BEGIN
	(*
	----------------------------------------------------------------------------------------
	|                                                                                      |
	|  Copyright  2023             FORTNA Europe BV                                        |
	|  All Rights Reserved         Netherlands                                             |
	|                                                                                      |
	----------------------------------------------------------------------------------------

	Version history:
	Date        | Version   | Author          | Remark
	----------------------------------------------------------------------------------------
	22/3/2022   | 0.1       | R. Golonka      | Unloader Alarm | DHL Munich 2023
	13/3/2024   | 0.2       | S.Nieswiec      | Alligned for new baseline
	*)

	REGION 1 - Jam
	    //  Program Alarm jam
	    #Jam(SIG := #iq_UDT_UnloaderStatus.Specific.PEC_EoS.Jam,
	         TIMESTAMP := #Time,
	         SD_1 := #is_ID);
	END_REGION

	REGION 2 - Disabled
	    //  Program Alarm disabled
	    #Disabled(SIG := #iq_UDT_UnloaderStatus.Specific.Disabled,
	              TIMESTAMP := #Time,
	              SD_1 := #is_ID);
	END_REGION

	REGION 3 - Too Long Parcel
	    //  Program Alarm too long parcel
	    #TooLongParcel(SIG := #iq_UDT_UnloaderStatus.Specific.TooLongParcel,
	                   TIMESTAMP := #Time,
	                   SD_1 := #is_ID);
	END_REGION

	REGION 4 - VFD Error
	    //  Program Alarm VFD Error
	    #VFDError(SIG := #iq_UDT_UnloaderStatus.Specific.VFDError,
	              TIMESTAMP := #Time,
	              SD_1 := #is_ID);
	END_REGION

	REGION 5 - Not healthy
	    //  Program Alarm not healthy
	    #NotHealthy(SIG := #iq_UDT_UnloaderStatus.Specific.NotHealthy,
	                TIMESTAMP := #Time,
	                SD_1 := #is_ID);
	END_REGION

END_FUNCTION_BLOCK

FUNCTION_BLOCK "FB_TP_ALARM_RIO"
{ S7_Optimized_Access := 'TRUE' }
VERSION : 0.1
// ATTRIBUTES
// AUTO_NUMBER = True
// BLOCK_NUMBER = 191
// END_ATTRIBUTES
   VAR_INPUT
      "Time" {InstructionName := 'DTL'; LibVersion := '1.0'; ExternalAccessible := 'False'; ExternalVisible := 'False'; ExternalWritable := 'False'} : DTL;   // Actual Time
      is_ID { ExternalAccessible := 'False'; ExternalVisible := 'False'; ExternalWritable := 'False'} : String;   // ID of component
   END_VAR

   VAR_IN_OUT
      iq_UDT_RIOStatus : "UDT_RIOStatus";   // Rio Status
   END_VAR

   VAR
      PNSlaveNotOnline {InstructionName := 'Program_Alarm'; LibVersion := '1.0'; ExternalAccessible := 'False'; ExternalVisible := 'False'; ExternalWritable := 'False'; S7_SetPoint := 'False'} : Program_Alarm;   // Program alarm profinet slave not online
      PNSlaveError {InstructionName := 'Program_Alarm'; LibVersion := '1.0'; ExternalAccessible := 'False'; ExternalVisible := 'False'; ExternalWritable := 'False'; S7_SetPoint := 'False'} : Program_Alarm;   // Program alarm profinet slave error
      ET200sp_ErrorModule {InstructionName := 'Program_Alarm'; LibVersion := '1.0'; ExternalAccessible := 'False'; ExternalVisible := 'False'; ExternalWritable := 'False'; S7_SetPoint := 'False'} : Array[0..31] of Program_Alarm;   // Program alarm ET200sp module error
      PNSlaveWarning {InstructionName := 'Program_Alarm'; LibVersion := '1.0'; ExternalAccessible := 'False'; ExternalVisible := 'False'; ExternalWritable := 'False'; S7_SetPoint := 'False'} : Program_Alarm;   // Program alarm profinet slave warning
   END_VAR

   VAR_TEMP
      ti_NrOfArrayEl : Int;   // Number of array element
      ti_ArraySize : Int;   // Array size
   END_VAR


BEGIN
	(*
	----------------------------------------------------------------------------------------
	|                                                                                      |
	|  Copyright  2023             FORTNA Europe BV                                        |
	|  All Rights Reserved         Netherlands                                             |
	|                                                                                      |
	----------------------------------------------------------------------------------------

	Version history:
	Date        | Version   | Author          | Remark
	----------------------------------------------------------------------------------------
	22/03/2023  | 0.1       | R. Golonka      | RIO Alarm | DHL Munich 2023
	13/3/2024   | 0.2       | S.Nieswiec      | Alligned for new baseline
	*)
	REGION 1 - Profinet slave not online
	    // Program alarm profinet slave not online
	    #PNSlaveNotOnline(SIG := #iq_UDT_RIOStatus.Specific.PNSlaveNotOnline,
	                      TIMESTAMP := #Time,
	                      SD_1 := #is_ID);
	END_REGION

	REGION 2 - Profinet slave error
	    // Program alarm profinet slave error
	    #PNSlaveError(SIG := #iq_UDT_RIOStatus.Specific.PNSlaveError,
	                  TIMESTAMP := #Time,
	                  SD_1 := #is_ID);
	END_REGION

	REGION 3 - Profinet slave warning
	    // Program alarm profinet slave warning
	    #PNSlaveWarning(SIG := #iq_UDT_RIOStatus.Specific.PNSlaveWarning,
	                    TIMESTAMP := #Time,
	                    SD_1 := #is_ID);
	END_REGION

	REGION 4 - ET200SP module error
	    // Array size
	    #ti_ArraySize := "FC_GetNrOfArrayEl"(#iq_UDT_RIOStatus.Specific.ET200sp_ErrorModule);

	    // Program alarm ET200SP module error
	    FOR #ti_NrOfArrayEl := 0 TO (#ti_ArraySize - 1) DO
	        #ET200sp_ErrorModule[#ti_NrOfArrayEl](SIG := #iq_UDT_RIOStatus.Specific.ET200sp_ErrorModule[#ti_NrOfArrayEl],
	                                              TIMESTAMP := #Time,
	                                              SD_1 := #is_ID);
	    END_FOR;
	END_REGION
END_FUNCTION_BLOCK

FUNCTION_BLOCK "FB_TP_ALARM_RetractableRoller"
{ S7_Optimized_Access := 'TRUE' }
VERSION : 0.1
// ATTRIBUTES
// AUTO_NUMBER = True
// BLOCK_NUMBER = 190
// END_ATTRIBUTES
   VAR_INPUT
      "Time" { ExternalAccessible := 'False'; ExternalVisible := 'False'; ExternalWritable := 'False'} : LDT;   // Actual Time
      is_ID { ExternalAccessible := 'False'; ExternalVisible := 'False'; ExternalWritable := 'False'} : String;   // ID of component
   END_VAR

   VAR_IN_OUT
      iq_UDT_RetractableRollerStatus : "UDT_RetractrableRoller_Status";
   END_VAR

   VAR
      NoHomePosition {InstructionName := 'Program_Alarm'; LibVersion := '1.0'; ExternalAccessible := 'False'; ExternalVisible := 'False'; ExternalWritable := 'False'; S7_SetPoint := 'False'} : Program_Alarm;
      RollerError {InstructionName := 'Program_Alarm'; LibVersion := '1.0'; ExternalAccessible := 'False'; ExternalVisible := 'False'; ExternalWritable := 'False'; S7_SetPoint := 'False'} : Program_Alarm;
   END_VAR


BEGIN
	(*
	----------------------------------------------------------------------------------------
	|                                                                                      |
	|  Copyright  2023             FORTNA Europe BV                                        |
	|  All Rights Reserved         Netherlands                                             |
	|                                                                                      |
	----------------------------------------------------------------------------------------

	Version history:
	Date        | Version   | Author          | Remark
	----------------------------------------------------------------------------------------
	09/05/2023   | 0.1       | M. Diebel       | ABSwitch Alarm | DHL Munich 2023
	13/3/2024    | 0.2       | S.Nieswiec      | Alligned for new baseline
	*)

	REGION 1 - NoHomePosition
	    //Program Alarm NoHomePosition
	    #NoHomePosition(SIG := #iq_UDT_RetractableRollerStatus.Specific.NoHomePosition,
	                    TIMESTAMP := #Time,
	                    SD_1 := #is_ID);
	END_REGION

	REGION 2 - RollerError
	    //Program Alarm RollerError
	    #RollerError(SIG := #iq_UDT_RetractableRollerStatus.Specific.RollerError,
	                 TIMESTAMP := #Time,
	                 SD_1 := #is_ID);
	END_REGION
END_FUNCTION_BLOCK

FUNCTION_BLOCK "FB_TP_ALARM_Rapiscan"
{ S7_Optimized_Access := 'TRUE' }
VERSION : 0.1
// ATTRIBUTES
// AUTO_NUMBER = True
// BLOCK_NUMBER = 189
// END_ATTRIBUTES
   VAR_INPUT
      "Time" { ExternalAccessible := 'False'; ExternalVisible := 'False'; ExternalWritable := 'False'} : LDT;   // Actual Time
      is_ID { ExternalAccessible := 'False'; ExternalVisible := 'False'; ExternalWritable := 'False'} : String;   // ID of component
   END_VAR

   VAR_IN_OUT
      iq_UDT_RapiscanStatus : "UDT_RapiscanStatus";   // Rapiscan Status
   END_VAR

   VAR
      XrayEnergised {InstructionName := 'Program_Alarm'; LibVersion := '1.0'; ExternalAccessible := 'False'; ExternalVisible := 'False'; ExternalWritable := 'False'; S7_SetPoint := 'False'} : Program_Alarm;   // Program Alarm Xray energised error
      XrayFault {InstructionName := 'Program_Alarm'; LibVersion := '1.0'; ExternalAccessible := 'False'; ExternalVisible := 'False'; ExternalWritable := 'False'; S7_SetPoint := 'False'} : Program_Alarm;   // Program Alarm Xray foult error
      XrayRdyRCV {InstructionName := 'Program_Alarm'; LibVersion := '1.0'; ExternalAccessible := 'False'; ExternalVisible := 'False'; ExternalWritable := 'False'; S7_SetPoint := 'False'} : Program_Alarm;   // Program Alarm Xray ready recieve info
      XrayRdySend {InstructionName := 'Program_Alarm'; LibVersion := '1.0'; ExternalAccessible := 'False'; ExternalVisible := 'False'; ExternalWritable := 'False'; S7_SetPoint := 'False'} : Program_Alarm;   // Program Alarm Xray ready send info
      BagScanning {InstructionName := 'Program_Alarm'; LibVersion := '1.0'; ExternalAccessible := 'False'; ExternalVisible := 'False'; ExternalWritable := 'False'; S7_SetPoint := 'False'} : Program_Alarm;   // Program Alarm bag scanming info
      TransportMode {InstructionName := 'Program_Alarm'; LibVersion := '1.0'; ExternalAccessible := 'False'; ExternalVisible := 'False'; ExternalWritable := 'False'; S7_SetPoint := 'False'} : Program_Alarm;   // Program Alarm transport mode info
      BackBelt {InstructionName := 'Program_Alarm'; LibVersion := '1.0'; ExternalAccessible := 'False'; ExternalVisible := 'False'; ExternalWritable := 'False'; S7_SetPoint := 'False'} : Program_Alarm;   // Program Alarm backbelt info
   END_VAR


BEGIN
	(*
	----------------------------------------------------------------------------------------
	|                                                                                      |
	|  Copyright  2023             FORTNA Europe BV                                        |
	|  All Rights Reserved         Netherlands                                             |
	|                                                                                      |
	----------------------------------------------------------------------------------------

	Version history:
	Date        | Version   | Author          | Remark
	----------------------------------------------------------------------------------------
	25/4/2022   | 1.0       | M. Diebel       | Rapiscan Alarm | DHL Munich 2023
	13/3/2024   | 1.1       | S.Nieswiec      | Alligned for new baseline
	*)

	REGION 1 - XrayEnergised
	    //Program Alarm Xray energised error
	    #XrayEnergised(SIG := #iq_UDT_RapiscanStatus.XraySpecific.XrayEnergised,
	                   TIMESTAMP := #Time,
	                   SD_1 := #is_ID);
	END_REGION

	REGION 2 - XrayFault
	    //Program Alarm Xray foult error
	    #XrayFault(SIG := #iq_UDT_RapiscanStatus.XraySpecific.XrayFault,
	               TIMESTAMP := #Time,
	               SD_1 := #is_ID);
	END_REGION

	REGION 3 - XrayRdyRCV
	    //Program Alarm Xray ready recieve info
	    #XrayRdyRCV(SIG := #iq_UDT_RapiscanStatus.XraySpecific.XrayRdyRCV,
	                TIMESTAMP := #Time,
	                SD_1 := #is_ID);
	END_REGION

	REGION 4 - XrayRdySend
	    //Program Alarm Xray ready send info
	    #XrayRdySend(SIG := #iq_UDT_RapiscanStatus.XraySpecific.XrayRdySend,
	                 TIMESTAMP := #Time,
	                 SD_1 := #is_ID);
	END_REGION

	REGION 5 - BagScanning
	    //Program Alarm bag scanming info
	    #BagScanning(SIG := #iq_UDT_RapiscanStatus.XraySpecific.BagScanning,
	                 TIMESTAMP := #Time,
	                 SD_1 := #is_ID);
	END_REGION

	REGION 6 - TransportMode
	    //Program Alarm transport mode info
	    #TransportMode(SIG := #iq_UDT_RapiscanStatus.XraySpecific.TransportMode,
	                   TIMESTAMP := #Time,
	                   SD_1 := #is_ID);
	END_REGION

	REGION 7 - BackBelt
	    //Program Alarm backbelt info
	    #BackBelt(SIG := #iq_UDT_RapiscanStatus.XraySpecific.BackBelt,
	              TIMESTAMP := #Time,
	              SD_1 := #is_ID);
	END_REGION



END_FUNCTION_BLOCK

FUNCTION_BLOCK "FB_TP_ALARM_PNNode"
{ S7_Optimized_Access := 'TRUE' }
VERSION : 0.1
// ATTRIBUTES
// AUTO_NUMBER = True
// BLOCK_NUMBER = 188
// END_ATTRIBUTES
   VAR_INPUT
      "Time" {InstructionName := 'DTL'; LibVersion := '1.0'; ExternalAccessible := 'False'; ExternalVisible := 'False'; ExternalWritable := 'False'} : DTL;   // Actual Time
      is_ID { ExternalAccessible := 'False'; ExternalVisible := 'False'; ExternalWritable := 'False'} : String;   // ID of component
   END_VAR

   VAR_IN_OUT
      iq_UDT_PNNode_Status : "UDT_PNNodeStatus";   // PNNode Status
   END_VAR

   VAR
      PNSlaveNotOnline {InstructionName := 'Program_Alarm'; LibVersion := '1.0'; ExternalAccessible := 'False'; ExternalVisible := 'False'; ExternalWritable := 'False'; S7_SetPoint := 'False'} : Program_Alarm;   // Program alarm profinet slave net online
      PNSlaveError {InstructionName := 'Program_Alarm'; LibVersion := '1.0'; ExternalAccessible := 'False'; ExternalVisible := 'False'; ExternalWritable := 'False'; S7_SetPoint := 'False'} : Program_Alarm;   // Program alarm profinet slave error
      PNSlaveWarning {InstructionName := 'Program_Alarm'; LibVersion := '1.0'; ExternalAccessible := 'False'; ExternalVisible := 'False'; ExternalWritable := 'False'; S7_SetPoint := 'False'} : Program_Alarm;   // Program alarm profinet slave warning
   END_VAR


BEGIN
	(*
	----------------------------------------------------------------------------------------
	|                                                                                      |
	|  Copyright  2023             FORTNA Europe BV                                        |
	|  All Rights Reserved         Netherlands                                             |
	|                                                                                      |
	----------------------------------------------------------------------------------------

	Version history:
	Date        | Version   | Author          | Remark
	----------------------------------------------------------------------------------------
	22/03/2023  | 0.1       | R. Golonka      | PN Node Alarm | DHL Munich 2023
	13/3/2024   | 0.2       | S.Nieswiec      | Alligned for new baseline
	*)

	REGION 1 - Profinet slave not online
	    // Program Alarm profinet slave not online
	    #PNSlaveNotOnline(SIG := #iq_UDT_PNNode_Status.Specific.PNSlaveNotOnline,
	                      TIMESTAMP := #Time,
	                      SD_1 := #is_ID);
	END_REGION

	REGION 2 - Profinet slave error
	    // Program Alarm profinet slave error
	    #PNSlaveError(SIG := #iq_UDT_PNNode_Status.Specific.PNSlaveError,
	                  TIMESTAMP := #Time,
	                  SD_1 := #is_ID);
	END_REGION

	REGION 3 - Profinet slave warning
	    // Program Alarm profinet slave warning
	    #PNSlaveWarning(SIG := #iq_UDT_PNNode_Status.Specific.PNSlaveWarning,
	                    TIMESTAMP := #Time,
	                    SD_1 := #is_ID);
	END_REGION
END_FUNCTION_BLOCK

FUNCTION_BLOCK "FB_TP_ALARM_PECUpdate"
{ S7_Optimized_Access := 'TRUE' }
VERSION : 0.1
// ATTRIBUTES
// AUTO_NUMBER = True
// BLOCK_NUMBER = 187
// END_ATTRIBUTES
   VAR_INPUT
      "Time" {InstructionName := 'DTL'; LibVersion := '1.0'; ExternalAccessible := 'False'; ExternalVisible := 'False'; ExternalWritable := 'False'} : DTL;   // Actual Time
      is_ID { ExternalAccessible := 'False'; ExternalVisible := 'False'; ExternalWritable := 'False'} : String;   // ID of component
   END_VAR

   VAR_IN_OUT
      iq_UDT_PECUpdate_Status : "UDT_PECUpdateStatus";   // PEC Update Status
   END_VAR

   VAR
      Jam {InstructionName := 'Program_Alarm'; LibVersion := '1.0'; ExternalAccessible := 'False'; ExternalVisible := 'False'; ExternalWritable := 'False'; S7_SetPoint := 'False'} : Program_Alarm;   // Program Alarm Jam
      TooManyLost {InstructionName := 'Program_Alarm'; LibVersion := '1.0'; ExternalAccessible := 'False'; ExternalVisible := 'False'; ExternalWritable := 'False'; S7_SetPoint := 'False'} : Program_Alarm;   // Program Alarm Too many losy
      LowPerformance {InstructionName := 'Program_Alarm'; LibVersion := '1.0'; ExternalAccessible := 'False'; ExternalVisible := 'False'; ExternalWritable := 'False'; S7_SetPoint := 'False'} : Program_Alarm;   // Program Alarm Low performance
   END_VAR


BEGIN
	(*
	----------------------------------------------------------------------------------------
	|                                                                                      |
	|  Copyright  2023             FORTNA Europe BV                                        |
	|  All Rights Reserved         Netherlands                                             |
	|                                                                                      |
	----------------------------------------------------------------------------------------

	Version history:
	Date        | Version   | Author          | Remark
	----------------------------------------------------------------------------------------
	22/3/2022   | 0.1       | R. Golonka      | PEC Update Alarm | DHL Munich 2023
	13/3/2024   | 0.2       | S.Nieswiec      | Alligned for new baseline
	*)

	REGION 1- Jam
	    // Program Alarm Jam
	    #Jam(SIG := #iq_UDT_PECUpdate_Status.Jam,
	         TIMESTAMP := #Time,
	         SD_1 := #is_ID);
	END_REGION

	REGION 2 - Too many lost
	    // Program Alarm Too many losy
	    #TooManyLost(SIG := #iq_UDT_PECUpdate_Status.TooManyLost,
	                 TIMESTAMP := #Time,
	                 SD_1 := #is_ID);
	END_REGION

	REGION 3 - Low Performance
	    // Program Alarm Low performance
	    #LowPerformance(SIG := #iq_UDT_PECUpdate_Status.LowPerformance,
	                    TIMESTAMP := #Time,
	                    SD_1 := #is_ID);
	END_REGION

END_FUNCTION_BLOCK

FUNCTION_BLOCK "FB_TP_ALARM_PEC"
{ S7_Optimized_Access := 'TRUE' }
VERSION : 0.1
// ATTRIBUTES
// AUTO_NUMBER = True
// BLOCK_NUMBER = 186
// END_ATTRIBUTES
   VAR_INPUT
      "Time" {InstructionName := 'DTL'; LibVersion := '1.0'; ExternalAccessible := 'False'; ExternalVisible := 'False'; ExternalWritable := 'False'} : DTL;   // Actual Time
      is_ID { ExternalAccessible := 'False'; ExternalVisible := 'False'; ExternalWritable := 'False'} : String;   // ID of component
   END_VAR

   VAR_IN_OUT
      iq_UDT_PEC_Status : "UDT_PECStatus";   // PEC Status
   END_VAR

   VAR
      Jam {InstructionName := 'Program_Alarm'; LibVersion := '1.0'; ExternalAccessible := 'False'; ExternalVisible := 'False'; ExternalWritable := 'False'; S7_SetPoint := 'False'} : Program_Alarm;   // Program Alarm Jam
   END_VAR


BEGIN
	(*
	----------------------------------------------------------------------------------------
	|                                                                                      |
	|  Copyright  2023             FORTNA Europe BV                                        |
	|  All Rights Reserved         Netherlands                                             |
	|                                                                                      |
	----------------------------------------------------------------------------------------

	Version history:
	Date        | Version   | Author          | Remark
	----------------------------------------------------------------------------------------
	22/3/2022   | 0.1       | R. Golonka      | PEC Alarm | DHL Munich 2023
	13/3/2024   | 0.2       | S.Nieswiec      | Alligned for new baseline
	*)

	REGION 1- Jam
	    // Program Alarm Jam
	    #Jam(SIG := #iq_UDT_PEC_Status.Jam,
	         TIMESTAMP := #Time,
	         SD_1 := #is_ID);
	END_REGION


END_FUNCTION_BLOCK

FUNCTION_BLOCK "FB_TP_ALARM_PDP"
{ S7_Optimized_Access := 'TRUE' }
VERSION : 0.1
// ATTRIBUTES
// AUTO_NUMBER = True
// BLOCK_NUMBER = 185
// END_ATTRIBUTES
   VAR_INPUT
      "Time" { ExternalAccessible := 'False'; ExternalVisible := 'False'; ExternalWritable := 'False'} : LDT;   // Actual Time
      is_ID { ExternalAccessible := 'False'; ExternalVisible := 'False'; ExternalWritable := 'False'} : String;   // ID of component
   END_VAR

   VAR_IN_OUT
      iq_UDT_PDPStatus : "UDT_PDPStatus";   // PDP Status
   END_VAR

   VAR
      CircuitBreakersTripped {InstructionName := 'Program_Alarm'; LibVersion := '1.0'; ExternalAccessible := 'False'; ExternalVisible := 'False'; ExternalWritable := 'False'; S7_SetPoint := 'False'} : Program_Alarm;   // Program Alarm circuit breakers tripped
      CircuitBreakerStateF100_F200_F300 {InstructionName := 'Program_Alarm'; LibVersion := '1.0'; ExternalAccessible := 'False'; ExternalVisible := 'False'; ExternalWritable := 'False'; S7_SetPoint := 'False'} : Program_Alarm;   // Program Alarm circuit breakers state
      CircuitBreakerStatePM {InstructionName := 'Program_Alarm'; LibVersion := '1.0'; ExternalAccessible := 'False'; ExternalVisible := 'False'; ExternalWritable := 'False'; S7_SetPoint := 'False'} : Program_Alarm;   // Program Alarm circuit breakers state PM
      CircuitBreakerTrippedF101 {InstructionName := 'Program_Alarm'; LibVersion := '1.0'; ExternalAccessible := 'False'; ExternalVisible := 'False'; ExternalWritable := 'False'; S7_SetPoint := 'False'} : Program_Alarm;   // Program Alarm circuit breakers tripped
      CircuitBreakerTrippedF102 {InstructionName := 'Program_Alarm'; LibVersion := '1.0'; ExternalAccessible := 'False'; ExternalVisible := 'False'; ExternalWritable := 'False'; S7_SetPoint := 'False'} : Program_Alarm;   // Program Alarm circuit breakers tripped
      CircuitBreakerTrippedF103 {InstructionName := 'Program_Alarm'; LibVersion := '1.0'; ExternalAccessible := 'False'; ExternalVisible := 'False'; ExternalWritable := 'False'; S7_SetPoint := 'False'} : Program_Alarm;   // Program Alarm circuit breakers tripped
      CircuitBreakerTrippedF104 {InstructionName := 'Program_Alarm'; LibVersion := '1.0'; ExternalAccessible := 'False'; ExternalVisible := 'False'; ExternalWritable := 'False'; S7_SetPoint := 'False'} : Program_Alarm;   // Program Alarm circuit breakers tripped
      CircuitBreakerTrippedF105 {InstructionName := 'Program_Alarm'; LibVersion := '1.0'; ExternalAccessible := 'False'; ExternalVisible := 'False'; ExternalWritable := 'False'; S7_SetPoint := 'False'} : Program_Alarm;   // Program Alarm circuit breakers tripped
      CircuitBreakerTrippedF106 {InstructionName := 'Program_Alarm'; LibVersion := '1.0'; ExternalAccessible := 'False'; ExternalVisible := 'False'; ExternalWritable := 'False'; S7_SetPoint := 'False'} : Program_Alarm;   // Program Alarm circuit breakers tripped
      CircuitBreakerTrippedF107 {InstructionName := 'Program_Alarm'; LibVersion := '1.0'; ExternalAccessible := 'False'; ExternalVisible := 'False'; ExternalWritable := 'False'; S7_SetPoint := 'False'} : Program_Alarm;   // Program Alarm circuit breakers tripped
      CircuitBreakerTrippedF108 {InstructionName := 'Program_Alarm'; LibVersion := '1.0'; ExternalAccessible := 'False'; ExternalVisible := 'False'; ExternalWritable := 'False'; S7_SetPoint := 'False'} : Program_Alarm;   // Program Alarm circuit breakers tripped
      CircuitBreakerTrippedF109 {InstructionName := 'Program_Alarm'; LibVersion := '1.0'; ExternalAccessible := 'False'; ExternalVisible := 'False'; ExternalWritable := 'False'; S7_SetPoint := 'False'} : Program_Alarm;   // Program Alarm circuit breakers tripped
      CircuitBreakerTrippedF110 {InstructionName := 'Program_Alarm'; LibVersion := '1.0'; ExternalAccessible := 'False'; ExternalVisible := 'False'; ExternalWritable := 'False'; S7_SetPoint := 'False'} : Program_Alarm;   // Program Alarm circuit breakers tripped
      CircuitBreakerTrippedF111 {InstructionName := 'Program_Alarm'; LibVersion := '1.0'; ExternalAccessible := 'False'; ExternalVisible := 'False'; ExternalWritable := 'False'; S7_SetPoint := 'False'} : Program_Alarm;   // Program Alarm circuit breakers tripped
      CircuitBreakerTrippedF112 {InstructionName := 'Program_Alarm'; LibVersion := '1.0'; ExternalAccessible := 'False'; ExternalVisible := 'False'; ExternalWritable := 'False'; S7_SetPoint := 'False'} : Program_Alarm;   // Program Alarm circuit breakers tripped
      CircuitBreakerTrippedF113 {InstructionName := 'Program_Alarm'; LibVersion := '1.0'; ExternalAccessible := 'False'; ExternalVisible := 'False'; ExternalWritable := 'False'; S7_SetPoint := 'False'} : Program_Alarm;   // Program Alarm circuit breakers tripped
      CircuitBreakerTrippedF114 {InstructionName := 'Program_Alarm'; LibVersion := '1.0'; ExternalAccessible := 'False'; ExternalVisible := 'False'; ExternalWritable := 'False'; S7_SetPoint := 'False'} : Program_Alarm;   // Program Alarm circuit breakers tripped
      CircuitBreakerTrippedF115 {InstructionName := 'Program_Alarm'; LibVersion := '1.0'; ExternalAccessible := 'False'; ExternalVisible := 'False'; ExternalWritable := 'False'; S7_SetPoint := 'False'} : Program_Alarm;   // Program Alarm circuit breakers tripped
      CircuitBreakerTrippedF116 {InstructionName := 'Program_Alarm'; LibVersion := '1.0'; ExternalAccessible := 'False'; ExternalVisible := 'False'; ExternalWritable := 'False'; S7_SetPoint := 'False'} : Program_Alarm;   // Program Alarm circuit breakers tripped
      CircuitBreakerTrippedF117 {InstructionName := 'Program_Alarm'; LibVersion := '1.0'; ExternalAccessible := 'False'; ExternalVisible := 'False'; ExternalWritable := 'False'; S7_SetPoint := 'False'} : Program_Alarm;   // Program Alarm circuit breakers tripped
      CircuitBreakerTrippedF118 {InstructionName := 'Program_Alarm'; LibVersion := '1.0'; ExternalAccessible := 'False'; ExternalVisible := 'False'; ExternalWritable := 'False'; S7_SetPoint := 'False'} : Program_Alarm;   // Program Alarm circuit breakers tripped
      CircuitBreakerTrippedF119 {InstructionName := 'Program_Alarm'; LibVersion := '1.0'; ExternalAccessible := 'False'; ExternalVisible := 'False'; ExternalWritable := 'False'; S7_SetPoint := 'False'} : Program_Alarm;   // Program Alarm circuit breakers tripped
      CircuitBreakerTrippedF120 {InstructionName := 'Program_Alarm'; LibVersion := '1.0'; ExternalAccessible := 'False'; ExternalVisible := 'False'; ExternalWritable := 'False'; S7_SetPoint := 'False'} : Program_Alarm;   // Program Alarm circuit breakers tripped
      CircuitBreakerTrippedF121 {InstructionName := 'Program_Alarm'; LibVersion := '1.0'; ExternalAccessible := 'False'; ExternalVisible := 'False'; ExternalWritable := 'False'; S7_SetPoint := 'False'} : Program_Alarm;   // Program Alarm circuit breakers tripped
      CircuitBreakerTrippedF122 {InstructionName := 'Program_Alarm'; LibVersion := '1.0'; ExternalAccessible := 'False'; ExternalVisible := 'False'; ExternalWritable := 'False'; S7_SetPoint := 'False'} : Program_Alarm;   // Program Alarm circuit breakers tripped
      CircuitBreakerTrippedF123 {InstructionName := 'Program_Alarm'; LibVersion := '1.0'; ExternalAccessible := 'False'; ExternalVisible := 'False'; ExternalWritable := 'False'; S7_SetPoint := 'False'} : Program_Alarm;   // Program Alarm circuit breakers tripped
      CircuitBreakerTrippedF124 {InstructionName := 'Program_Alarm'; LibVersion := '1.0'; ExternalAccessible := 'False'; ExternalVisible := 'False'; ExternalWritable := 'False'; S7_SetPoint := 'False'} : Program_Alarm;   // Program Alarm circuit breakers tripped
      CircuitBreakerTrippedF125 {InstructionName := 'Program_Alarm'; LibVersion := '1.0'; ExternalAccessible := 'False'; ExternalVisible := 'False'; ExternalWritable := 'False'; S7_SetPoint := 'False'} : Program_Alarm;   // Program Alarm circuit breakers tripped
      CircuitBreakerTrippedF126 {InstructionName := 'Program_Alarm'; LibVersion := '1.0'; ExternalAccessible := 'False'; ExternalVisible := 'False'; ExternalWritable := 'False'; S7_SetPoint := 'False'} : Program_Alarm;   // Program Alarm circuit breakers tripped
      CircuitBreakerTrippedF127 {InstructionName := 'Program_Alarm'; LibVersion := '1.0'; ExternalAccessible := 'False'; ExternalVisible := 'False'; ExternalWritable := 'False'; S7_SetPoint := 'False'} : Program_Alarm;   // Program Alarm circuit breakers tripped
      CircuitBreakerTrippedF128 {InstructionName := 'Program_Alarm'; LibVersion := '1.0'; ExternalAccessible := 'False'; ExternalVisible := 'False'; ExternalWritable := 'False'; S7_SetPoint := 'False'} : Program_Alarm;   // Program Alarm circuit breakers tripped
      CircuitBreakerTrippedF129 {InstructionName := 'Program_Alarm'; LibVersion := '1.0'; ExternalAccessible := 'False'; ExternalVisible := 'False'; ExternalWritable := 'False'; S7_SetPoint := 'False'} : Program_Alarm;   // Program Alarm circuit breakers tripped
      CircuitBreakerTrippedF130 {InstructionName := 'Program_Alarm'; LibVersion := '1.0'; ExternalAccessible := 'False'; ExternalVisible := 'False'; ExternalWritable := 'False'; S7_SetPoint := 'False'} : Program_Alarm;   // Program Alarm circuit breakers tripped
      CircuitBreakerTrippedF131 {InstructionName := 'Program_Alarm'; LibVersion := '1.0'; ExternalAccessible := 'False'; ExternalVisible := 'False'; ExternalWritable := 'False'; S7_SetPoint := 'False'} : Program_Alarm;   // Program Alarm circuit breakers tripped
      CircuitBreakerTrippedF132 {InstructionName := 'Program_Alarm'; LibVersion := '1.0'; ExternalAccessible := 'False'; ExternalVisible := 'False'; ExternalWritable := 'False'; S7_SetPoint := 'False'} : Program_Alarm;   // Program Alarm circuit breakers tripped
      CircuitBreakerTrippedF133 {InstructionName := 'Program_Alarm'; LibVersion := '1.0'; ExternalAccessible := 'False'; ExternalVisible := 'False'; ExternalWritable := 'False'; S7_SetPoint := 'False'} : Program_Alarm;   // Program Alarm circuit breakers tripped
      CircuitBreakerTrippedF134 {InstructionName := 'Program_Alarm'; LibVersion := '1.0'; ExternalAccessible := 'False'; ExternalVisible := 'False'; ExternalWritable := 'False'; S7_SetPoint := 'False'} : Program_Alarm;   // Program Alarm circuit breakers tripped
      CircuitBreakerTrippedF135 {InstructionName := 'Program_Alarm'; LibVersion := '1.0'; ExternalAccessible := 'False'; ExternalVisible := 'False'; ExternalWritable := 'False'; S7_SetPoint := 'False'} : Program_Alarm;   // Program Alarm circuit breakers tripped
      CircuitBreakerTrippedF201 {InstructionName := 'Program_Alarm'; LibVersion := '1.0'; ExternalAccessible := 'False'; ExternalVisible := 'False'; ExternalWritable := 'False'; S7_SetPoint := 'False'} : Program_Alarm;   // Program Alarm circuit breakers tripped
      CircuitBreakerTrippedF202 {InstructionName := 'Program_Alarm'; LibVersion := '1.0'; ExternalAccessible := 'False'; ExternalVisible := 'False'; ExternalWritable := 'False'; S7_SetPoint := 'False'} : Program_Alarm;   // Program Alarm circuit breakers tripped
      CircuitBreakerTrippedF203 {InstructionName := 'Program_Alarm'; LibVersion := '1.0'; ExternalAccessible := 'False'; ExternalVisible := 'False'; ExternalWritable := 'False'; S7_SetPoint := 'False'} : Program_Alarm;   // Program Alarm circuit breakers tripped
      CircuitBreakerTrippedF204 {InstructionName := 'Program_Alarm'; LibVersion := '1.0'; ExternalAccessible := 'False'; ExternalVisible := 'False'; ExternalWritable := 'False'; S7_SetPoint := 'False'} : Program_Alarm;   // Program Alarm circuit breakers tripped
      CircuitBreakerTrippedF205 {InstructionName := 'Program_Alarm'; LibVersion := '1.0'; ExternalAccessible := 'False'; ExternalVisible := 'False'; ExternalWritable := 'False'; S7_SetPoint := 'False'} : Program_Alarm;   // Program Alarm circuit breakers tripped
      CircuitBreakerTrippedF206 {InstructionName := 'Program_Alarm'; LibVersion := '1.0'; ExternalAccessible := 'False'; ExternalVisible := 'False'; ExternalWritable := 'False'; S7_SetPoint := 'False'} : Program_Alarm;   // Program Alarm circuit breakers tripped
      CircuitBreakerTrippedF207 {InstructionName := 'Program_Alarm'; LibVersion := '1.0'; ExternalAccessible := 'False'; ExternalVisible := 'False'; ExternalWritable := 'False'; S7_SetPoint := 'False'} : Program_Alarm;   // Program Alarm circuit breakers tripped
      CircuitBreakerTrippedF208 {InstructionName := 'Program_Alarm'; LibVersion := '1.0'; ExternalAccessible := 'False'; ExternalVisible := 'False'; ExternalWritable := 'False'; S7_SetPoint := 'False'} : Program_Alarm;   // Program Alarm circuit breakers tripped
      CircuitBreakerTrippedF209 {InstructionName := 'Program_Alarm'; LibVersion := '1.0'; ExternalAccessible := 'False'; ExternalVisible := 'False'; ExternalWritable := 'False'; S7_SetPoint := 'False'} : Program_Alarm;   // Program Alarm circuit breakers tripped
      CircuitBreakerTrippedF210 {InstructionName := 'Program_Alarm'; LibVersion := '1.0'; ExternalAccessible := 'False'; ExternalVisible := 'False'; ExternalWritable := 'False'; S7_SetPoint := 'False'} : Program_Alarm;   // Program Alarm circuit breakers tripped
      CircuitBreakerTrippedF211 {InstructionName := 'Program_Alarm'; LibVersion := '1.0'; ExternalAccessible := 'False'; ExternalVisible := 'False'; ExternalWritable := 'False'; S7_SetPoint := 'False'} : Program_Alarm;   // Program Alarm circuit breakers tripped
      CircuitBreakerTrippedF212 {InstructionName := 'Program_Alarm'; LibVersion := '1.0'; ExternalAccessible := 'False'; ExternalVisible := 'False'; ExternalWritable := 'False'; S7_SetPoint := 'False'} : Program_Alarm;   // Program Alarm circuit breakers tripped
      CircuitBreakerTrippedF213 {InstructionName := 'Program_Alarm'; LibVersion := '1.0'; ExternalAccessible := 'False'; ExternalVisible := 'False'; ExternalWritable := 'False'; S7_SetPoint := 'False'} : Program_Alarm;   // Program Alarm circuit breakers tripped
      CircuitBreakerTrippedF214 {InstructionName := 'Program_Alarm'; LibVersion := '1.0'; ExternalAccessible := 'False'; ExternalVisible := 'False'; ExternalWritable := 'False'; S7_SetPoint := 'False'} : Program_Alarm;   // Program Alarm circuit breakers tripped
      CircuitBreakerTrippedF215 {InstructionName := 'Program_Alarm'; LibVersion := '1.0'; ExternalAccessible := 'False'; ExternalVisible := 'False'; ExternalWritable := 'False'; S7_SetPoint := 'False'} : Program_Alarm;   // Program Alarm circuit breakers tripped
      CircuitBreakerTrippedF216 {InstructionName := 'Program_Alarm'; LibVersion := '1.0'; ExternalAccessible := 'False'; ExternalVisible := 'False'; ExternalWritable := 'False'; S7_SetPoint := 'False'} : Program_Alarm;   // Program Alarm circuit breakers tripped
      CircuitBreakerTrippedF217 {InstructionName := 'Program_Alarm'; LibVersion := '1.0'; ExternalAccessible := 'False'; ExternalVisible := 'False'; ExternalWritable := 'False'; S7_SetPoint := 'False'} : Program_Alarm;   // Program Alarm circuit breakers tripped
      CircuitBreakerTrippedF218 {InstructionName := 'Program_Alarm'; LibVersion := '1.0'; ExternalAccessible := 'False'; ExternalVisible := 'False'; ExternalWritable := 'False'; S7_SetPoint := 'False'} : Program_Alarm;   // Program Alarm circuit breakers tripped
      CircuitBreakerTrippedF219 {InstructionName := 'Program_Alarm'; LibVersion := '1.0'; ExternalAccessible := 'False'; ExternalVisible := 'False'; ExternalWritable := 'False'; S7_SetPoint := 'False'} : Program_Alarm;   // Program Alarm circuit breakers tripped
      CircuitBreakerTrippedF220 {InstructionName := 'Program_Alarm'; LibVersion := '1.0'; ExternalAccessible := 'False'; ExternalVisible := 'False'; ExternalWritable := 'False'; S7_SetPoint := 'False'} : Program_Alarm;   // Program Alarm circuit breakers tripped
      CircuitBreakerTrippedF221 {InstructionName := 'Program_Alarm'; LibVersion := '1.0'; ExternalAccessible := 'False'; ExternalVisible := 'False'; ExternalWritable := 'False'; S7_SetPoint := 'False'} : Program_Alarm;   // Program Alarm circuit breakers tripped
      CircuitBreakerTrippedF222 {InstructionName := 'Program_Alarm'; LibVersion := '1.0'; ExternalAccessible := 'False'; ExternalVisible := 'False'; ExternalWritable := 'False'; S7_SetPoint := 'False'} : Program_Alarm;   // Program Alarm circuit breakers tripped
      CircuitBreakerTrippedF223 {InstructionName := 'Program_Alarm'; LibVersion := '1.0'; ExternalAccessible := 'False'; ExternalVisible := 'False'; ExternalWritable := 'False'; S7_SetPoint := 'False'} : Program_Alarm;   // Program Alarm circuit breakers tripped
      CircuitBreakerTrippedF224 {InstructionName := 'Program_Alarm'; LibVersion := '1.0'; ExternalAccessible := 'False'; ExternalVisible := 'False'; ExternalWritable := 'False'; S7_SetPoint := 'False'} : Program_Alarm;   // Program Alarm circuit breakers tripped
      CircuitBreakerTrippedF225 {InstructionName := 'Program_Alarm'; LibVersion := '1.0'; ExternalAccessible := 'False'; ExternalVisible := 'False'; ExternalWritable := 'False'; S7_SetPoint := 'False'} : Program_Alarm;   // Program Alarm circuit breakers tripped
      CircuitBreakerTrippedF226 {InstructionName := 'Program_Alarm'; LibVersion := '1.0'; ExternalAccessible := 'False'; ExternalVisible := 'False'; ExternalWritable := 'False'; S7_SetPoint := 'False'} : Program_Alarm;   // Program Alarm circuit breakers tripped
      CircuitBreakerTrippedF227 {InstructionName := 'Program_Alarm'; LibVersion := '1.0'; ExternalAccessible := 'False'; ExternalVisible := 'False'; ExternalWritable := 'False'; S7_SetPoint := 'False'} : Program_Alarm;   // Program Alarm circuit breakers tripped
      CircuitBreakerTrippedF228 {InstructionName := 'Program_Alarm'; LibVersion := '1.0'; ExternalAccessible := 'False'; ExternalVisible := 'False'; ExternalWritable := 'False'; S7_SetPoint := 'False'} : Program_Alarm;   // Program Alarm circuit breakers tripped
      CircuitBreakerTrippedF229 {InstructionName := 'Program_Alarm'; LibVersion := '1.0'; ExternalAccessible := 'False'; ExternalVisible := 'False'; ExternalWritable := 'False'; S7_SetPoint := 'False'} : Program_Alarm;   // Program Alarm circuit breakers tripped
      CircuitBreakerTrippedF501 {InstructionName := 'Program_Alarm'; LibVersion := '1.0'; ExternalAccessible := 'False'; ExternalVisible := 'False'; ExternalWritable := 'False'; S7_SetPoint := 'False'} : Program_Alarm;   // Program Alarm circuit breakers tripped
      CircuitBreakerTrippedF502 {InstructionName := 'Program_Alarm'; LibVersion := '1.0'; ExternalAccessible := 'False'; ExternalVisible := 'False'; ExternalWritable := 'False'; S7_SetPoint := 'False'} : Program_Alarm;   // Program Alarm circuit breakers tripped
      CircuitBreakerTrippedF503 {InstructionName := 'Program_Alarm'; LibVersion := '1.0'; ExternalAccessible := 'False'; ExternalVisible := 'False'; ExternalWritable := 'False'; S7_SetPoint := 'False'} : Program_Alarm;   // Program Alarm circuit breakers tripped
      CircuitBreakerTrippedF504 {InstructionName := 'Program_Alarm'; LibVersion := '1.0'; ExternalAccessible := 'False'; ExternalVisible := 'False'; ExternalWritable := 'False'; S7_SetPoint := 'False'} : Program_Alarm;   // Program Alarm circuit breakers tripped
      CircuitBreakerTrippedF505 {InstructionName := 'Program_Alarm'; LibVersion := '1.0'; ExternalAccessible := 'False'; ExternalVisible := 'False'; ExternalWritable := 'False'; S7_SetPoint := 'False'} : Program_Alarm;   // Program Alarm circuit breakers tripped
      CircuitBreakerTrippedF506 {InstructionName := 'Program_Alarm'; LibVersion := '1.0'; ExternalAccessible := 'False'; ExternalVisible := 'False'; ExternalWritable := 'False'; S7_SetPoint := 'False'} : Program_Alarm;   // Program Alarm circuit breakers tripped
      CircuitBreakerTrippedF507 {InstructionName := 'Program_Alarm'; LibVersion := '1.0'; ExternalAccessible := 'False'; ExternalVisible := 'False'; ExternalWritable := 'False'; S7_SetPoint := 'False'} : Program_Alarm;   // Program Alarm circuit breakers tripped
      CircuitBreakerTrippedF508 {InstructionName := 'Program_Alarm'; LibVersion := '1.0'; ExternalAccessible := 'False'; ExternalVisible := 'False'; ExternalWritable := 'False'; S7_SetPoint := 'False'} : Program_Alarm;   // Program Alarm circuit breakers tripped
      CircuitBreakerTrippedF509 {InstructionName := 'Program_Alarm'; LibVersion := '1.0'; ExternalAccessible := 'False'; ExternalVisible := 'False'; ExternalWritable := 'False'; S7_SetPoint := 'False'} : Program_Alarm;   // Program Alarm circuit breakers tripped
      CircuitBreakerTrippedF510 {InstructionName := 'Program_Alarm'; LibVersion := '1.0'; ExternalAccessible := 'False'; ExternalVisible := 'False'; ExternalWritable := 'False'; S7_SetPoint := 'False'} : Program_Alarm;   // Program Alarm circuit breakers tripped
      CircuitBreakerTrippedF511 {InstructionName := 'Program_Alarm'; LibVersion := '1.0'; ExternalAccessible := 'False'; ExternalVisible := 'False'; ExternalWritable := 'False'; S7_SetPoint := 'False'} : Program_Alarm;   // Program Alarm circuit breakers tripped
      CircuitBreakerTrippedF512 {InstructionName := 'Program_Alarm'; LibVersion := '1.0'; ExternalAccessible := 'False'; ExternalVisible := 'False'; ExternalWritable := 'False'; S7_SetPoint := 'False'} : Program_Alarm;   // Program Alarm circuit breakers tripped
   END_VAR


BEGIN
	(*
	----------------------------------------------------------------------------------------
	|                                                                                      |
	|  Copyright  2023             FORTNA Europe BV                                        |
	|  All Rights Reserved         Netherlands                                             |
	|                                                                                      |
	----------------------------------------------------------------------------------------

	Version history:
	Date        | Version   | Author          | Remark
	----------------------------------------------------------------------------------------
	24/04/2022   | 0.1       | M.Diebel       | PDP Alarm | DHL Munich 2023
	24/07/2023   | 0.2       | R.Golonka      | PDP Alarm update F130-F135
	13/3/2024    | 0.3       | S.Nieswiec      | Alligned for new baseline
	*)

	REGION 1 - Circuit breakers tripped
	    //Program alarm circuit breakers tripped
	    #CircuitBreakersTripped(SIG := #iq_UDT_PDPStatus.Specific.CircuitBreakersTripped,
	                            TIMESTAMP := #Time,
	                            SD_1 := #is_ID);
	END_REGION


	REGION 2 - CircuitBreakerState F100_F200_F300
	    //Program alarm Circuit Breaker State F100 F200 F300
	    #CircuitBreakerStateF100_F200_F300(SIG := #iq_UDT_PDPStatus.Specific.CircuitBreakerStateF100_F200_F300,
	                                       TIMESTAMP := #Time,
	                                       SD_1 := #is_ID);
	END_REGION

	REGION 3 - CircuitBreakerStatPM
	    //Program alarm Circuit Breaker Stat PM
	    #CircuitBreakerStatePM(SIG := #iq_UDT_PDPStatus.Specific.CircuitBreakerStatePM,
	                           TIMESTAMP := #Time,
	                           SD_1 := #is_ID);
	END_REGION

	REGION 4 - CircuitBreakerTrippedF101
	    //Program alarm Circuit Breaker Tripped F101
	    #CircuitBreakerTrippedF101(SIG := #iq_UDT_PDPStatus.Specific.CircuitBreakerTrippedF101,
	                               TIMESTAMP := #Time,
	                               SD_1 := #is_ID);
	END_REGION

	REGION 5 - CircuitBreakerTrippedF102
	    //Program alarm Circuit Breaker Tripped F102
	    #CircuitBreakerTrippedF102(SIG := #iq_UDT_PDPStatus.Specific.CircuitBreakerTrippedF102,
	                               TIMESTAMP := #Time,
	                               SD_1 := #is_ID);
	END_REGION

	REGION 6 - CircuitBreakerTrippedF103
	    //Program alarm Circuit Breaker Tripped F103
	    #CircuitBreakerTrippedF103(SIG := #iq_UDT_PDPStatus.Specific.CircuitBreakerTrippedF103,
	                               TIMESTAMP := #Time,
	                               SD_1 := #is_ID);
	END_REGION

	REGION 7 - CircuitBreakerTrippedF104
	    //Program alarm Circuit Breaker Tripped F104
	    #CircuitBreakerTrippedF104(SIG := #iq_UDT_PDPStatus.Specific.CircuitBreakerTrippedF104,
	                               TIMESTAMP := #Time,
	                               SD_1 := #is_ID);
	END_REGION

	REGION 8 - CircuitBreakerTrippedF105
	    //Program alarm Circuit Breaker Tripped F105
	    #CircuitBreakerTrippedF105(SIG := #iq_UDT_PDPStatus.Specific.CircuitBreakerTrippedF105,
	                               TIMESTAMP := #Time,
	                               SD_1 := #is_ID);
	END_REGION

	REGION 9 - CircuitBreakerTrippedF106
	    //Program alarm Circuit Breaker Tripped F106
	    #CircuitBreakerTrippedF106(SIG := #iq_UDT_PDPStatus.Specific.CircuitBreakerTrippedF106,
	                               TIMESTAMP := #Time,
	                               SD_1 := #is_ID);
	END_REGION

	REGION 10 - CircuitBreakerTrippedF107
	    //Program alarm Circuit Breaker Tripped F107
	    #CircuitBreakerTrippedF107(SIG := #iq_UDT_PDPStatus.Specific.CircuitBreakerTrippedF107,
	                               TIMESTAMP := #Time,
	                               SD_1 := #is_ID);
	END_REGION

	REGION 11 - CircuitBreakerTrippedF108
	    //Program alarm Circuit Breaker Tripped F108
	    #CircuitBreakerTrippedF108(SIG := #iq_UDT_PDPStatus.Specific.CircuitBreakerTrippedF108,
	                               TIMESTAMP := #Time,
	                               SD_1 := #is_ID);
	END_REGION

	REGION 12 - CircuitBreakerTrippedF109
	    //Program alarm Circuit Breaker Tripped F109
	    #CircuitBreakerTrippedF109(SIG := #iq_UDT_PDPStatus.Specific.CircuitBreakerTrippedF109,
	                               TIMESTAMP := #Time,
	                               SD_1 := #is_ID);
	END_REGION

	REGION 13 - CircuitBreakerTrippedF110
	    //Program alarm Circuit Breaker Tripped F110
	    #CircuitBreakerTrippedF110(SIG := #iq_UDT_PDPStatus.Specific.CircuitBreakerTrippedF110,
	                               TIMESTAMP := #Time,
	                               SD_1 := #is_ID);
	END_REGION

	REGION 14 - CircuitBreakerTrippedF111
	    //Program alarm Circuit Breaker Tripped F111
	    #CircuitBreakerTrippedF111(SIG := #iq_UDT_PDPStatus.Specific.CircuitBreakerTrippedF111,
	                               TIMESTAMP := #Time,
	                               SD_1 := #is_ID);
	END_REGION

	REGION 15 - CircuitBreakerTrippedF112
	    //Program alarm Circuit Breaker Tripped F112
	    #CircuitBreakerTrippedF112(SIG := #iq_UDT_PDPStatus.Specific.CircuitBreakerTrippedF112,
	                               TIMESTAMP := #Time,
	                               SD_1 := #is_ID);
	END_REGION

	REGION 16 - CircuitBreakerTrippedF113
	    //Program alarm Circuit Breaker Tripped F113
	    #CircuitBreakerTrippedF113(SIG := #iq_UDT_PDPStatus.Specific.CircuitBreakerTrippedF113,
	                               TIMESTAMP := #Time,
	                               SD_1 := #is_ID);
	END_REGION

	REGION 17 - CircuitBreakerTrippedF114
	    //Program alarm Circuit Breaker Tripped F114
	    #CircuitBreakerTrippedF114(SIG := #iq_UDT_PDPStatus.Specific.CircuitBreakerTrippedF114,
	                               TIMESTAMP := #Time,
	                               SD_1 := #is_ID);
	END_REGION

	REGION 18 - CircuitBreakerTrippedF115
	    //Program alarm Circuit Breaker Tripped F115
	    #CircuitBreakerTrippedF115(SIG := #iq_UDT_PDPStatus.Specific.CircuitBreakerTrippedF115,
	                               TIMESTAMP := #Time,
	                               SD_1 := #is_ID);
	END_REGION

	REGION 19 - CircuitBreakerTrippedF116
	    //Program alarm Circuit Breaker Tripped F116
	    #CircuitBreakerTrippedF116(SIG := #iq_UDT_PDPStatus.Specific.CircuitBreakerTrippedF116,
	                               TIMESTAMP := #Time,
	                               SD_1 := #is_ID);
	END_REGION

	REGION 20 - CircuitBreakerTrippedF117
	    //Program alarm Circuit Breaker Tripped F117
	    #CircuitBreakerTrippedF117(SIG := #iq_UDT_PDPStatus.Specific.CircuitBreakerTrippedF117,
	                               TIMESTAMP := #Time,
	                               SD_1 := #is_ID);
	END_REGION

	REGION 21 - CircuitBreakerTrippedF118
	    //Program alarm Circuit Breaker Tripped F118
	    #CircuitBreakerTrippedF118(SIG := #iq_UDT_PDPStatus.Specific.CircuitBreakerTrippedF118,
	                               TIMESTAMP := #Time,
	                               SD_1 := #is_ID);
	END_REGION

	REGION 22 - CircuitBreakerTrippedF119
	    //Program alarm Circuit Breaker Tripped F119
	    #CircuitBreakerTrippedF119(SIG := #iq_UDT_PDPStatus.Specific.CircuitBreakerTrippedF119,
	                               TIMESTAMP := #Time,
	                               SD_1 := #is_ID);
	END_REGION

	REGION 23 - CircuitBreakerTrippedF120
	    //Program alarm Circuit Breaker Tripped F120
	    #CircuitBreakerTrippedF120(SIG := #iq_UDT_PDPStatus.Specific.CircuitBreakerTrippedF120,
	                               TIMESTAMP := #Time,
	                               SD_1 := #is_ID);
	END_REGION

	REGION 24 - CircuitBreakerTrippedF121
	    //Program alarm Circuit Breaker Tripped F121
	    #CircuitBreakerTrippedF121(SIG := #iq_UDT_PDPStatus.Specific.CircuitBreakerTrippedF121,
	                               TIMESTAMP := #Time,
	                               SD_1 := #is_ID);
	END_REGION

	REGION 25 - CircuitBreakerTrippedF122
	    //Program alarm Circuit Breaker Tripped F122
	    #CircuitBreakerTrippedF122(SIG := #iq_UDT_PDPStatus.Specific.CircuitBreakerTrippedF122,
	                               TIMESTAMP := #Time,
	                               SD_1 := #is_ID);
	END_REGION

	REGION 26 - CircuitBreakerTrippedF123
	    //Program alarm Circuit Breaker Tripped F123
	    #CircuitBreakerTrippedF123(SIG := #iq_UDT_PDPStatus.Specific.CircuitBreakerTrippedF123,
	                               TIMESTAMP := #Time,
	                               SD_1 := #is_ID);
	END_REGION

	REGION 27 - CircuitBreakerTrippedF124
	    //Program alarm Circuit Breaker Tripped F124
	    #CircuitBreakerTrippedF124(SIG := #iq_UDT_PDPStatus.Specific.CircuitBreakerTrippedF124,
	                               TIMESTAMP := #Time,
	                               SD_1 := #is_ID);
	END_REGION

	REGION 28 - CircuitBreakerTrippedF125
	    //Program alarm Circuit Breaker Tripped F125
	    #CircuitBreakerTrippedF125(SIG := #iq_UDT_PDPStatus.Specific.CircuitBreakerTrippedF125,
	                               TIMESTAMP := #Time,
	                               SD_1 := #is_ID);
	END_REGION

	REGION 29 - CircuitBreakerTrippedF126
	    //Program alarm Circuit Breaker Tripped F126
	    #CircuitBreakerTrippedF126(SIG := #iq_UDT_PDPStatus.Specific.CircuitBreakerTrippedF126,
	                               TIMESTAMP := #Time,
	                               SD_1 := #is_ID);
	END_REGION

	REGION 30 - CircuitBreakerTrippedF127
	    //Program alarm Circuit Breaker Tripped F127
	    #CircuitBreakerTrippedF127(SIG := #iq_UDT_PDPStatus.Specific.CircuitBreakerTrippedF127,
	                               TIMESTAMP := #Time,
	                               SD_1 := #is_ID);
	END_REGION

	REGION 31 - CircuitBreakerTrippedF128
	    //Program alarm Circuit Breaker Tripped F128
	    #CircuitBreakerTrippedF128(SIG := #iq_UDT_PDPStatus.Specific.CircuitBreakerTrippedF128,
	                               TIMESTAMP := #Time,
	                               SD_1 := #is_ID);
	END_REGION

	REGION 32 - CircuitBreakerTrippedF129
	    //Program alarm Circuit Breaker Tripped F129
	    #CircuitBreakerTrippedF129(SIG := #iq_UDT_PDPStatus.Specific.CircuitBreakerTrippedF129,
	                               TIMESTAMP := #Time,
	                               SD_1 := #is_ID);
	END_REGION

	REGION 33 - CircuitBreakerTrippedF201
	    //Program alarm Circuit Breaker Tripped F201
	    #CircuitBreakerTrippedF201(SIG := #iq_UDT_PDPStatus.Specific.CircuitBreakerTrippedF201,
	                               TIMESTAMP := #Time,
	                               SD_1 := #is_ID);
	END_REGION

	REGION 34 - CircuitBreakerTrippedF202
	    //Program alarm Circuit Breaker Tripped F102
	    #CircuitBreakerTrippedF202(SIG := #iq_UDT_PDPStatus.Specific.CircuitBreakerTrippedF202,
	                               TIMESTAMP := #Time,
	                               SD_1 := #is_ID);
	END_REGION

	REGION 35 - CircuitBreakerTrippedF203
	    //Program alarm Circuit Breaker Tripped F203
	    #CircuitBreakerTrippedF203(SIG := #iq_UDT_PDPStatus.Specific.CircuitBreakerTrippedF203,
	                               TIMESTAMP := #Time,
	                               SD_1 := #is_ID);
	END_REGION

	REGION 36 - CircuitBreakerTripped2104
	    //Program alarm Circuit Breaker Tripped F204
	    #CircuitBreakerTrippedF204(SIG := #iq_UDT_PDPStatus.Specific.CircuitBreakerTrippedF204,
	                               TIMESTAMP := #Time,
	                               SD_1 := #is_ID);
	END_REGION

	REGION 37 - CircuitBreakerTrippedF205
	    //Program alarm Circuit Breaker Tripped F205
	    #CircuitBreakerTrippedF205(SIG := #iq_UDT_PDPStatus.Specific.CircuitBreakerTrippedF205,
	                               TIMESTAMP := #Time,
	                               SD_1 := #is_ID);
	END_REGION

	REGION 38 - CircuitBreakerTrippedF206
	    //Program alarm Circuit Breaker Tripped F206
	    #CircuitBreakerTrippedF206(SIG := #iq_UDT_PDPStatus.Specific.CircuitBreakerTrippedF206,
	                               TIMESTAMP := #Time,
	                               SD_1 := #is_ID);
	END_REGION

	REGION 39 - CircuitBreakerTrippedF207
	    //Program alarm Circuit Breaker Tripped F207
	    #CircuitBreakerTrippedF207(SIG := #iq_UDT_PDPStatus.Specific.CircuitBreakerTrippedF207,
	                               TIMESTAMP := #Time,
	                               SD_1 := #is_ID);
	END_REGION

	REGION 40 - CircuitBreakerTrippedF208
	    //Program alarm Circuit Breaker Tripped F208
	    #CircuitBreakerTrippedF208(SIG := #iq_UDT_PDPStatus.Specific.CircuitBreakerTrippedF208,
	                               TIMESTAMP := #Time,
	                               SD_1 := #is_ID);
	END_REGION

	REGION 41 - CircuitBreakerTrippedF209
	    //Program alarm Circuit Breaker Tripped F209
	    #CircuitBreakerTrippedF209(SIG := #iq_UDT_PDPStatus.Specific.CircuitBreakerTrippedF209,
	                               TIMESTAMP := #Time,
	                               SD_1 := #is_ID);
	END_REGION

	REGION 42 - CircuitBreakerTrippedF210
	    //Program alarm Circuit Breaker Tripped F210
	    #CircuitBreakerTrippedF210(SIG := #iq_UDT_PDPStatus.Specific.CircuitBreakerTrippedF210,
	                               TIMESTAMP := #Time,
	                               SD_1 := #is_ID);
	END_REGION

	REGION 43 - CircuitBreakerTrippedF211
	    //Program alarm Circuit Breaker Tripped F211
	    #CircuitBreakerTrippedF211(SIG := #iq_UDT_PDPStatus.Specific.CircuitBreakerTrippedF211,
	                               TIMESTAMP := #Time,
	                               SD_1 := #is_ID);
	END_REGION

	REGION 44 - CircuitBreakerTrippedF212
	    //Program alarm Circuit Breaker Tripped F212
	    #CircuitBreakerTrippedF212(SIG := #iq_UDT_PDPStatus.Specific.CircuitBreakerTrippedF212,
	                               TIMESTAMP := #Time,
	                               SD_1 := #is_ID);
	END_REGION

	REGION 45 - CircuitBreakerTrippedF213
	    //Program alarm Circuit Breaker Tripped F213
	    #CircuitBreakerTrippedF213(SIG := #iq_UDT_PDPStatus.Specific.CircuitBreakerTrippedF213,
	                               TIMESTAMP := #Time,
	                               SD_1 := #is_ID);
	END_REGION

	REGION 46 - CircuitBreakerTrippedF214
	    //Program alarm Circuit Breaker Tripped F214
	    #CircuitBreakerTrippedF214(SIG := #iq_UDT_PDPStatus.Specific.CircuitBreakerTrippedF214,
	                               TIMESTAMP := #Time,
	                               SD_1 := #is_ID);
	END_REGION

	REGION 47 - CircuitBreakerTrippedF215
	    //Program alarm Circuit Breaker Tripped F215
	    #CircuitBreakerTrippedF215(SIG := #iq_UDT_PDPStatus.Specific.CircuitBreakerTrippedF215,
	                               TIMESTAMP := #Time,
	                               SD_1 := #is_ID);
	END_REGION

	REGION 48 - CircuitBreakerTrippedF216
	    //Program alarm Circuit Breaker Tripped F216
	    #CircuitBreakerTrippedF216(SIG := #iq_UDT_PDPStatus.Specific.CircuitBreakerTrippedF216,
	                               TIMESTAMP := #Time,
	                               SD_1 := #is_ID);
	END_REGION

	REGION 49 - CircuitBreakerTrippedF217
	    //Program alarm Circuit Breaker Tripped F217
	    #CircuitBreakerTrippedF217(SIG := #iq_UDT_PDPStatus.Specific.CircuitBreakerTrippedF217,
	                               TIMESTAMP := #Time,
	                               SD_1 := #is_ID);
	END_REGION

	REGION 50 - CircuitBreakerTrippedF218
	    //Program alarm Circuit Breaker Tripped F218
	    #CircuitBreakerTrippedF218(SIG := #iq_UDT_PDPStatus.Specific.CircuitBreakerTrippedF218,
	                               TIMESTAMP := #Time,
	                               SD_1 := #is_ID);
	END_REGION

	REGION 51 - CircuitBreakerTrippedF219
	    //Program alarm Circuit Breaker Tripped F219
	    #CircuitBreakerTrippedF219(SIG := #iq_UDT_PDPStatus.Specific.CircuitBreakerTrippedF219,
	                               TIMESTAMP := #Time,
	                               SD_1 := #is_ID);
	END_REGION

	REGION 52 - CircuitBreakerTrippedF220
	    //Program alarm Circuit Breaker Tripped F220
	    #CircuitBreakerTrippedF220(SIG := #iq_UDT_PDPStatus.Specific.CircuitBreakerTrippedF220,
	                               TIMESTAMP := #Time,
	                               SD_1 := #is_ID);
	END_REGION

	REGION 53 - CircuitBreakerTrippedF121
	    //Program alarm Circuit Breaker Tripped F221
	    #CircuitBreakerTrippedF221(SIG := #iq_UDT_PDPStatus.Specific.CircuitBreakerTrippedF221,
	                               TIMESTAMP := #Time,
	                               SD_1 := #is_ID);
	END_REGION

	REGION 54 - CircuitBreakerTrippedF222
	    //Program alarm Circuit Breaker Tripped F222
	    #CircuitBreakerTrippedF222(SIG := #iq_UDT_PDPStatus.Specific.CircuitBreakerTrippedF222,
	                               TIMESTAMP := #Time,
	                               SD_1 := #is_ID);
	END_REGION

	REGION 55 - CircuitBreakerTrippedF223
	    //Program alarm Circuit Breaker Tripped F223
	    #CircuitBreakerTrippedF223(SIG := #iq_UDT_PDPStatus.Specific.CircuitBreakerTrippedF223,
	                               TIMESTAMP := #Time,
	                               SD_1 := #is_ID);
	END_REGION

	REGION 56 - CircuitBreakerTrippedF224
	    //Program alarm Circuit Breaker Tripped F224
	    #CircuitBreakerTrippedF224(SIG := #iq_UDT_PDPStatus.Specific.CircuitBreakerTrippedF224,
	                               TIMESTAMP := #Time,
	                               SD_1 := #is_ID);
	END_REGION

	REGION 57 - CircuitBreakerTrippedF225
	    //Program alarm Circuit Breaker Tripped F225
	    #CircuitBreakerTrippedF225(SIG := #iq_UDT_PDPStatus.Specific.CircuitBreakerTrippedF225,
	                               TIMESTAMP := #Time,
	                               SD_1 := #is_ID);
	END_REGION

	REGION 58 - CircuitBreakerTrippedF226
	    //Program alarm Circuit Breaker Tripped F226
	    #CircuitBreakerTrippedF226(SIG := #iq_UDT_PDPStatus.Specific.CircuitBreakerTrippedF226,
	                               TIMESTAMP := #Time,
	                               SD_1 := #is_ID);
	END_REGION

	REGION 59 - CircuitBreakerTrippedF227
	    //Program alarm Circuit Breaker Tripped F227
	    #CircuitBreakerTrippedF227(SIG := #iq_UDT_PDPStatus.Specific.CircuitBreakerTrippedF227,
	                               TIMESTAMP := #Time,
	                               SD_1 := #is_ID);
	END_REGION

	REGION 60 - CircuitBreakerTrippedF228
	    //Program alarm Circuit Breaker Tripped F228
	    #CircuitBreakerTrippedF228(SIG := #iq_UDT_PDPStatus.Specific.CircuitBreakerTrippedF228,
	                               TIMESTAMP := #Time,
	                               SD_1 := #is_ID);
	END_REGION

	REGION 61 - CircuitBreakerTrippedF229
	    //Program alarm Circuit Breaker Tripped F229
	    #CircuitBreakerTrippedF229(SIG := #iq_UDT_PDPStatus.Specific.CircuitBreakerTrippedF229,
	                               TIMESTAMP := #Time,
	                               SD_1 := #is_ID);
	END_REGION

	REGION 62 - CircuitBreakerTrippedF501
	    //Program alarm Circuit Breaker Tripped F501
	    #CircuitBreakerTrippedF501(SIG := #iq_UDT_PDPStatus.Specific.CircuitBreakerTrippedF501,
	                               TIMESTAMP := #Time,
	                               SD_1 := #is_ID);
	END_REGION

	REGION 63 - CircuitBreakerTrippedF502
	    //Program alarm Circuit Breaker Tripped F502
	    #CircuitBreakerTrippedF502(SIG := #iq_UDT_PDPStatus.Specific.CircuitBreakerTrippedF502,
	                               TIMESTAMP := #Time,
	                               SD_1 := #is_ID);
	END_REGION

	REGION 64 - CircuitBreakerTrippedF503
	    //Program alarm Circuit Breaker Tripped F503
	    #CircuitBreakerTrippedF503(SIG := #iq_UDT_PDPStatus.Specific.CircuitBreakerTrippedF503,
	                               TIMESTAMP := #Time,
	                               SD_1 := #is_ID);
	END_REGION

	REGION 65 - CircuitBreakerTripped504
	    //Program alarm Circuit Breaker Tripped F504
	    #CircuitBreakerTrippedF504(SIG := #iq_UDT_PDPStatus.Specific.CircuitBreakerTrippedF504,
	                               TIMESTAMP := #Time,
	                               SD_1 := #is_ID);
	END_REGION

	REGION 66 - CircuitBreakerTrippedF505
	    //Program alarm Circuit Breaker Tripped F505
	    #CircuitBreakerTrippedF505(SIG := #iq_UDT_PDPStatus.Specific.CircuitBreakerTrippedF505,
	                               TIMESTAMP := #Time,
	                               SD_1 := #is_ID);
	END_REGION

	REGION 67 - CircuitBreakerTrippedF506
	    //Program alarm Circuit Breaker Tripped F506
	    #CircuitBreakerTrippedF506(SIG := #iq_UDT_PDPStatus.Specific.CircuitBreakerTrippedF506,
	                               TIMESTAMP := #Time,
	                               SD_1 := #is_ID);
	END_REGION

	REGION 68 - CircuitBreakerTrippedF507
	    //Program alarm Circuit Breaker Tripped F507
	    #CircuitBreakerTrippedF507(SIG := #iq_UDT_PDPStatus.Specific.CircuitBreakerTrippedF507,
	                               TIMESTAMP := #Time,
	                               SD_1 := #is_ID);
	END_REGION

	REGION 69 - CircuitBreakerTrippedF508
	    //Program alarm Circuit Breaker Tripped F508
	    #CircuitBreakerTrippedF508(SIG := #iq_UDT_PDPStatus.Specific.CircuitBreakerTrippedF508,
	                               TIMESTAMP := #Time,
	                               SD_1 := #is_ID);
	END_REGION

	REGION 70 - CircuitBreakerTrippedF509
	    //Program alarm Circuit Breaker Tripped F509
	    #CircuitBreakerTrippedF509(SIG := #iq_UDT_PDPStatus.Specific.CircuitBreakerTrippedF509,
	                               TIMESTAMP := #Time,
	                               SD_1 := #is_ID);
	END_REGION

	REGION 71 - CircuitBreakerTrippedF510
	    //Program alarm Circuit Breaker Tripped F510
	    #CircuitBreakerTrippedF510(SIG := #iq_UDT_PDPStatus.Specific.CircuitBreakerTrippedF510,
	                               TIMESTAMP := #Time,
	                               SD_1 := #is_ID);
	END_REGION

	REGION 72 - CircuitBreakerTrippedF511
	    //Program alarm Circuit Breaker Tripped F511
	    #CircuitBreakerTrippedF511(SIG := #iq_UDT_PDPStatus.Specific.CircuitBreakerTrippedF511,
	                               TIMESTAMP := #Time,
	                               SD_1 := #is_ID);
	END_REGION

	REGION 73 - CircuitBreakerTrippedF512
	    //Program alarm Circuit Breaker Tripped F512
	    #CircuitBreakerTrippedF512(SIG := #iq_UDT_PDPStatus.Specific.CircuitBreakerTrippedF512,
	                               TIMESTAMP := #Time,
	                               SD_1 := #is_ID);
	END_REGION

	REGION 74 - CircuitBreakerTrippedF130
	    //Program alarm Circuit Breaker Tripped F130
	    #CircuitBreakerTrippedF130(SIG := #iq_UDT_PDPStatus.Specific.CircuitBreakerTrippedF130,
	                               TIMESTAMP := #Time,
	                               SD_1 := #is_ID);
	END_REGION

	REGION 75 - CircuitBreakerTrippedF131
	    //Program alarm Circuit Breaker Tripped F131
	    #CircuitBreakerTrippedF131(SIG := #iq_UDT_PDPStatus.Specific.CircuitBreakerTrippedF131,
	                               TIMESTAMP := #Time,
	                               SD_1 := #is_ID);
	END_REGION

	REGION 76 - CircuitBreakerTrippedF132
	    //Program alarm Circuit Breaker Tripped F132
	    #CircuitBreakerTrippedF132(SIG := #iq_UDT_PDPStatus.Specific.CircuitBreakerTrippedF132,
	                               TIMESTAMP := #Time,
	                               SD_1 := #is_ID);
	END_REGION

	REGION 77 - CircuitBreakerTrippedF133
	    //Program alarm Circuit Breaker Tripped F133
	    #CircuitBreakerTrippedF133(SIG := #iq_UDT_PDPStatus.Specific.CircuitBreakerTrippedF133,
	                               TIMESTAMP := #Time,
	                               SD_1 := #is_ID);
	END_REGION

	REGION 78 - CircuitBreakerTrippedF134
	    //Program alarm Circuit Breaker Tripped F134
	    #CircuitBreakerTrippedF134(SIG := #iq_UDT_PDPStatus.Specific.CircuitBreakerTrippedF134,
	                               TIMESTAMP := #Time,
	                               SD_1 := #is_ID);
	END_REGION

	REGION 79 - CircuitBreakerTrippedF135
	    //Program alarm Circuit Breaker Tripped F135
	    #CircuitBreakerTrippedF135(SIG := #iq_UDT_PDPStatus.Specific.CircuitBreakerTrippedF135,
	                               TIMESTAMP := #Time,
	                               SD_1 := #is_ID);
	END_REGION

END_FUNCTION_BLOCK

FUNCTION_BLOCK "FB_TP_ALARM_Outfeed2States"
{ S7_Optimized_Access := 'TRUE' }
VERSION : 0.1
// ATTRIBUTES
// AUTO_NUMBER = True
// BLOCK_NUMBER = 184
// END_ATTRIBUTES
   VAR_INPUT
      "Time" { ExternalAccessible := 'False'; ExternalVisible := 'False'; ExternalWritable := 'False'} : LDT;   // Actual Time
      is_ID { ExternalAccessible := 'False'; ExternalVisible := 'False'; ExternalWritable := 'False'} : String;   // ID of component
   END_VAR

   VAR_IN_OUT
      iq_UDT_Outfeed2StatesStatus : "UDT_Outfeed2StatesStatus";   // Outfeed2states status
   END_VAR

   VAR
      ChuteFull {InstructionName := 'Program_Alarm'; LibVersion := '1.0'; ExternalAccessible := 'False'; ExternalVisible := 'False'; ExternalWritable := 'False'; S7_SetPoint := 'False'} : Program_Alarm;   // Program Alarm Chute Full
      ChuteHalfFull {InstructionName := 'Program_Alarm'; LibVersion := '1.0'; ExternalAccessible := 'False'; ExternalVisible := 'False'; ExternalWritable := 'False'; S7_SetPoint := 'False'} : Program_Alarm;   // Program Alarm Chute Half Full
      ChuteDisabled {InstructionName := 'Program_Alarm'; LibVersion := '1.0'; ExternalAccessible := 'False'; ExternalVisible := 'False'; ExternalWritable := 'False'; S7_SetPoint := 'False'} : Program_Alarm;   // Program Alarm Chute Disabled
   END_VAR


BEGIN
	(*
	----------------------------------------------------------------------------------------
	|                                                                                      |
	|  Copyright  2023             FORTNA Europe BV                                        |
	|  All Rights Reserved         Netherlands                                             |
	|                                                                                      |
	----------------------------------------------------------------------------------------

	Version history:
	Date        | Version   | Author          | Remark
	----------------------------------------------------------------------------------------
	22/3/2022   | 0.1       | R. Golonka      | Outfeed2States Alarm | DHL Munich 2023
	13/3/2024   | 0.2       | S.Nieswiec      | Alligned for new baseline
	*)

	REGION 1 - Chute Full
	    //  Program Alarm Chute full
	    #ChuteFull(SIG := #iq_UDT_Outfeed2StatesStatus.Specific.ChuteFull,
	               TIMESTAMP := #Time,
	               SD_1 := #is_ID);
	END_REGION

	REGION 2 - Chute Half Full
	    //  Program Alarm chute half full
	    #ChuteHalfFull(SIG := #iq_UDT_Outfeed2StatesStatus.Specific.ChuteHalfFull,
	                   TIMESTAMP := #Time,
	                   SD_1 := #is_ID);
	END_REGION

	REGION 3 - Chute Disabled
	    //  Program Alarm chute disabled
	    #ChuteDisabled(SIG := #iq_UDT_Outfeed2StatesStatus.Specific.ChuteDisabled,
	                   TIMESTAMP := #Time,
	                   SD_1 := #is_ID);
	END_REGION
END_FUNCTION_BLOCK

FUNCTION_BLOCK "FB_TP_ALARM_NORD_VFD"
{ S7_Optimized_Access := 'TRUE' }
VERSION : 0.1
// ATTRIBUTES
// AUTO_NUMBER = True
// BLOCK_NUMBER = 183
// END_ATTRIBUTES
   VAR_INPUT
      "Time" {InstructionName := 'DTL'; LibVersion := '1.0'; ExternalAccessible := 'False'; ExternalVisible := 'False'; ExternalWritable := 'False'} : DTL;   // Actual Time
      is_ID { ExternalAccessible := 'False'; ExternalVisible := 'False'; ExternalWritable := 'False'} : String;   // ID of component
      i_UDT_TP_Interface { ExternalAccessible := 'False'; ExternalVisible := 'False'; ExternalWritable := 'False'} : "UDT_TPInterfaceV2";   // HMI Interface
   END_VAR

   VAR_IN_OUT
      iq_UDT_VFD_Status : "UDT_VfdStatus";   // VFD status
   END_VAR

   VAR
      CommunicationErrorMovikit {InstructionName := 'Program_Alarm'; LibVersion := '1.0'; ExternalAccessible := 'False'; ExternalVisible := 'False'; ExternalWritable := 'False'; S7_SetPoint := 'False'} : Program_Alarm;   // Program Alarm communication error Movikit
      InternalVFDError {InstructionName := 'Program_Alarm'; LibVersion := '1.0'; ExternalAccessible := 'False'; ExternalVisible := 'False'; ExternalWritable := 'False'; S7_SetPoint := 'False'} : Program_Alarm;   // Program Alarm internal VFD error
      InternalVFDWarning {InstructionName := 'Program_Alarm'; LibVersion := '1.0'; ExternalAccessible := 'False'; ExternalVisible := 'False'; ExternalWritable := 'False'; S7_SetPoint := 'False'} : Program_Alarm;   // Program Alarm internal VFD Warning
      PNSlaveError {InstructionName := 'Program_Alarm'; LibVersion := '1.0'; ExternalAccessible := 'False'; ExternalVisible := 'False'; ExternalWritable := 'False'; S7_SetPoint := 'False'} : Program_Alarm;   // Program Alarm profinet slave error
      PNSlaveNotonline {InstructionName := 'Program_Alarm'; LibVersion := '1.0'; ExternalAccessible := 'False'; ExternalVisible := 'False'; ExternalWritable := 'False'; S7_SetPoint := 'False'} : Program_Alarm;   // Program Alarm profinet slave not online
      PNSlaveWarnnig {InstructionName := 'Program_Alarm'; LibVersion := '1.0'; ExternalAccessible := 'False'; ExternalVisible := 'False'; ExternalWritable := 'False'; S7_SetPoint := 'False'} : Program_Alarm;   // Program Alarm internal VFD Warning
      VFDRunningFeedbackError {InstructionName := 'Program_Alarm'; LibVersion := '1.0'; ExternalAccessible := 'False'; ExternalVisible := 'False'; ExternalWritable := 'False'; S7_SetPoint := 'False'} : Program_Alarm;   // Program Alarm VFD Feedback Error
      sx_AlarmCodeChange { ExternalAccessible := 'False'; ExternalVisible := 'False'; ExternalWritable := 'False'} : Bool;   // Alarm error code change trigger
      si_PreviousErrorCode { ExternalAccessible := 'False'; ExternalVisible := 'False'; ExternalWritable := 'False'} : Int;   // Previous error code
      sx_InternalErrorTrigger { ExternalAccessible := 'False'; ExternalVisible := 'False'; ExternalWritable := 'False'} : Bool;   // Internal error trigger
      sx_InternalWarningTrigger { ExternalAccessible := 'False'; ExternalVisible := 'False'; ExternalWritable := 'False'} : Bool;   // Internal warning trigger
      ss_ErrorCode { ExternalAccessible := 'False'; ExternalVisible := 'False'; ExternalWritable := 'False'} : String;   // Nord error code number
      si_ErrorCode { ExternalAccessible := 'False'; ExternalVisible := 'False'; ExternalWritable := 'False'} : Int;
   END_VAR

   VAR_TEMP
      ts_ErrorText : String;   // Temp. Error text
      ts_ErrorTextGerman : String;   // Temp. german error text
   END_VAR


BEGIN
	(*
	----------------------------------------------------------------------------------------
	|                                                                                      |
	|  Copyright  2023             FORTNA Europe BV                                        |
	|  All Rights Reserved         Netherlands                                             |
	|                                                                                      |
	----------------------------------------------------------------------------------------

	Version history:
	Date        | Version   | Author          | Remark
	----------------------------------------------------------------------------------------
	22/03/2023  | 0.1       | R. Golonka      | VFD NORD Alarm | DHL Munich 2023
	30/01/2023  | 0.2       | R. Golonka      | VFD NORD error code
	                                          | need to be genereted in both language on the trigger <--------- !!!
	13/3/2024   | 0.3       | S.Nieswiec      | Alligned for new baseline
	*)

	REGION 1- Communiation Error
	    // Program Alarm communication error Movikit
	    #CommunicationErrorMovikit(SIG := #iq_UDT_VFD_Status.CommunicationErrorMovikit,
	                               TIMESTAMP := #Time,
	                               SD_1 := #is_ID);
	END_REGION

	REGION 2 - Alarm change trigger
	    // Alarm change
	    #sx_AlarmCodeChange := (#si_PreviousErrorCode <> #iq_UDT_VFD_Status.ErrorCode);
	    // Previous alarm change
	    #si_PreviousErrorCode := #iq_UDT_VFD_Status.ErrorCode;
	    // Internal error trigger
	    #sx_InternalErrorTrigger := NOT #sx_AlarmCodeChange AND #iq_UDT_VFD_Status.InternalError;
	    // Internal warning trigger
	    #sx_InternalWarningTrigger := NOT #sx_AlarmCodeChange AND #iq_UDT_VFD_Status.InternalWarning;

	END_REGION

	REGION 4 - Error code with sub error code

	    #si_ErrorCode := (#iq_UDT_VFD_Status.ErrorCode * 10) + #iq_UDT_VFD_Status.SubErrorCode;

	END_REGION

	REGION 3- Error code to floating point string
	    // Nord system error code (like in Nord drive manual)
	    #ss_ErrorCode := '';
	    VAL_STRG(IN := #si_ErrorCode,
	             SIZE := 0,
	             PREC := 1,
	             FORMAT := 0,
	             P := 1,
	             OUT => #ss_ErrorCode);
	END_REGION

	REGION 4 - Eror text english

	    // Clear temporary string
	    #ts_ErrorText := '';

	    // Posibly error code
	    IF #sx_InternalErrorTrigger OR #sx_InternalWarningTrigger THEN
	        CASE #si_ErrorCode OF
	                // Error code to string code
	            10:
	                #ts_ErrorText := CONCAT(IN1 := 'Inverter overtemperature, error code: ', IN2 := #ss_ErrorCode);
	            11:
	                #ts_ErrorText := CONCAT(IN1 := 'Internal FI overtemperature, error code: ', IN2 := #ss_ErrorCode);
	            20:
	                #ts_ErrorText := CONCAT(IN1 := 'Motor overtemp.PTC, error code: ', IN2 := #ss_ErrorCode);
	            21:
	                #ts_ErrorText := CONCAT(IN1 := 'Motor overtemp.I²t, error code: ', IN2 := #ss_ErrorCode);
	            22:
	                #ts_ErrorText := CONCAT(IN1 := 'Ext Resistor Temp, error code: ', IN2 := #ss_ErrorCode);
	            30:
	                #ts_ErrorText := CONCAT(IN1 := 'Overcurrent I²t-Lim., error code: ', IN2 := #ss_ErrorCode);
	            31:
	                #ts_ErrorText := CONCAT(IN1 := 'Overcurrent Chopper, error code: ', IN2 := #ss_ErrorCode);
	            32:
	                #ts_ErrorText := CONCAT(IN1 := 'Overcurrent IGBT, error code: ', IN2 := #ss_ErrorCode);
	            33:
	                #ts_ErrorText := CONCAT(IN1 := 'Overcurrent IGBTfast, error code: ', IN2 := #ss_ErrorCode);
	            40:
	                #ts_ErrorText := CONCAT(IN1 := 'Module overcurrent, error code: ', IN2 := #ss_ErrorCode);
	            41:
	                #ts_ErrorText := CONCAT(IN1 := 'Overcurrent measurem, error code: ', IN2 := #ss_ErrorCode);
	            50:
	                #ts_ErrorText := CONCAT(IN1 := 'Overvoltage Ud, error code: ', IN2 := #ss_ErrorCode);
	            51:
	                #ts_ErrorText := CONCAT(IN1 := 'Mains overvoltage, error code: ', IN2 := #ss_ErrorCode);
	            60:
	                #ts_ErrorText := CONCAT(IN1 := 'Charging error, error code: ', IN2 := #ss_ErrorCode);
	            61:
	                #ts_ErrorText := CONCAT(IN1 := 'Mains low voltage, error code: ', IN2 := #ss_ErrorCode);
	            70:
	                #ts_ErrorText := CONCAT(IN1 := 'Mains Phase Failure, error code: ', IN2 := #ss_ErrorCode);
	            71:
	                #ts_ErrorText := CONCAT(IN1 := 'Phasefailure dc-link, error code: ', IN2 := #ss_ErrorCode);
	            80:
	                #ts_ErrorText := CONCAT(IN1 := 'Parameter lost, error code: ', IN2 := #ss_ErrorCode);
	            81:
	                #ts_ErrorText := CONCAT(IN1 := 'Inverter ID error, error code: ', IN2 := #ss_ErrorCode);
	            82:
	                #ts_ErrorText := CONCAT(IN1 := 'Reserved, error code: ', IN2 := #ss_ErrorCode);
	            83:
	                #ts_ErrorText := CONCAT(IN1 := 'Extern. EEPROM error, error code: ', IN2 := #ss_ErrorCode);
	            84:
	                #ts_ErrorText := CONCAT(IN1 := 'EEPROM intern. error, error code: ', IN2 := #ss_ErrorCode);
	            87:
	                #ts_ErrorText := CONCAT(IN1 := 'EEPROM copy differs, error code: ', IN2 := #ss_ErrorCode);
	            100:
	                #ts_ErrorText := CONCAT(IN1 := 'Bus time-out, error code: ', IN2 := #ss_ErrorCode);
	            101:
	                #ts_ErrorText := CONCAT(IN1 := 'System-error option, error code: ', IN2 := #ss_ErrorCode);
	            102:
	                #ts_ErrorText := CONCAT(IN1 := 'Bus time-out option, error code: ', IN2 := #ss_ErrorCode);
	            103:
	                #ts_ErrorText := CONCAT(IN1 := 'System-error option, error code: ', IN2 := #ss_ErrorCode);
	            104:
	                #ts_ErrorText := CONCAT(IN1 := 'Init-error option, error code: ', IN2 := #ss_ErrorCode);
	            105:
	                #ts_ErrorText := CONCAT(IN1 := 'System-error option, error code: ', IN2 := #ss_ErrorCode);
	            106:
	                #ts_ErrorText := CONCAT(IN1 := 'System-error option, error code: ', IN2 := #ss_ErrorCode);
	            107:
	                #ts_ErrorText := CONCAT(IN1 := 'System-error option, error code: ', IN2 := #ss_ErrorCode);
	            109:
	                #ts_ErrorText := CONCAT(IN1 := 'Missing Option /P120, error code: ', IN2 := #ss_ErrorCode);
	            110:
	                #ts_ErrorText := CONCAT(IN1 := 'Control terminals, error code: ', IN2 := #ss_ErrorCode);
	            120:
	                #ts_ErrorText := CONCAT(IN1 := 'External Watchdog, error code: ', IN2 := #ss_ErrorCode);
	            121:
	                #ts_ErrorText := CONCAT(IN1 := 'Limit moto./Customer, error code: ', IN2 := #ss_ErrorCode);
	            122:
	                #ts_ErrorText := CONCAT(IN1 := 'Limit gen., error code: ', IN2 := #ss_ErrorCode);
	            123:
	                #ts_ErrorText := CONCAT(IN1 := 'Torque Limit, error code: ', IN2 := #ss_ErrorCode);
	            124:
	                #ts_ErrorText := CONCAT(IN1 := 'Current limit, error code: ', IN2 := #ss_ErrorCode);
	            125:
	                #ts_ErrorText := CONCAT(IN1 := 'Load monitor, error code: ', IN2 := #ss_ErrorCode);
	            128:
	                #ts_ErrorText := CONCAT(IN1 := 'AI minimum, error code: ', IN2 := #ss_ErrorCode);
	            129:
	                #ts_ErrorText := CONCAT(IN1 := 'AI maximum, error code: ', IN2 := #ss_ErrorCode);
	            130:
	                #ts_ErrorText := CONCAT(IN1 := 'Encoder error, error code: ', IN2 := #ss_ErrorCode);
	            131:
	                #ts_ErrorText := CONCAT(IN1 := 'Speed slip error, error code: ', IN2 := #ss_ErrorCode);
	            132:
	                #ts_ErrorText := CONCAT(IN1 := 'Disconnect. control, error code: ', IN2 := #ss_ErrorCode);
	            160:
	                #ts_ErrorText := CONCAT(IN1 := 'Motor Phase Failure, error code: ', IN2 := #ss_ErrorCode);
	            161:
	                #ts_ErrorText := CONCAT(IN1 := 'Magn. Current Watch, error code: ', IN2 := #ss_ErrorCode);
	            180:
	                #ts_ErrorText := CONCAT(IN1 := 'Safety circuit, error code: ', IN2 := #ss_ErrorCode);
	            190:
	                #ts_ErrorText := CONCAT(IN1 := 'Parameter ident., error code: ', IN2 := #ss_ErrorCode);
	            191:
	                #ts_ErrorText := CONCAT(IN1 := 'Star Delta incorrect, error code: ', IN2 := #ss_ErrorCode);
	            200:
	                #ts_ErrorText := CONCAT(IN1 := 'Reserved, error code: ', IN2 := #ss_ErrorCode);
	            201:
	                #ts_ErrorText := CONCAT(IN1 := 'Watchdog, error code: ', IN2 := #ss_ErrorCode);
	            202:
	                #ts_ErrorText := CONCAT(IN1 := 'Stack overflow, error code: ', IN2 := #ss_ErrorCode);
	            203:
	                #ts_ErrorText := CONCAT(IN1 := 'Stack underflow, error code: ', IN2 := #ss_ErrorCode);
	            204:
	                #ts_ErrorText := CONCAT(IN1 := 'Undefined opcode, error code: ', IN2 := #ss_ErrorCode);
	            205:
	                #ts_ErrorText := CONCAT(IN1 := 'Protected Instruct., error code: ', IN2 := #ss_ErrorCode);
	            206:
	                #ts_ErrorText := CONCAT(IN1 := 'Illegal word Access, error code: ', IN2 := #ss_ErrorCode);
	            207:
	                #ts_ErrorText := CONCAT(IN1 := 'Illegal inst. Acces, error code: ', IN2 := #ss_ErrorCode);
	            208:
	                #ts_ErrorText := CONCAT(IN1 := 'Program memory error, error code: ', IN2 := #ss_ErrorCode);
	            209:
	                #ts_ErrorText := CONCAT(IN1 := 'Dual-ported RAM, error code: ', IN2 := #ss_ErrorCode);
	            210:
	                #ts_ErrorText := CONCAT(IN1 := 'NMI error, error code: ', IN2 := #ss_ErrorCode);
	            211:
	                #ts_ErrorText := CONCAT(IN1 := 'PLL error, error code: ', IN2 := #ss_ErrorCode);
	            212:
	                #ts_ErrorText := CONCAT(IN1 := 'ADU error, error code: ', IN2 := #ss_ErrorCode);
	            213:
	                #ts_ErrorText := CONCAT(IN1 := 'PMI error, error code: ', IN2 := #ss_ErrorCode);
	            214:
	                #ts_ErrorText := CONCAT(IN1 := 'Userstack overflow, error code: ', IN2 := #ss_ErrorCode);
	            ELSE  // Unknow alarm code
	                #ts_ErrorText := CONCAT(IN1 := 'Alarm unknown, error code: ', IN2 := (#ss_ErrorCode));
	        END_CASE;
	    ELSE
	        #ts_ErrorText := 'Alarm code change';
	    END_IF;

	    // Write error code
	    IF #sx_InternalErrorTrigger THEN
	        #ts_ErrorText := CONCAT(IN1 := #is_ID, IN2 := ' NORD VFD has internal error:', IN3 := #ts_ErrorText);
	    END_IF;

	    IF #sx_InternalWarningTrigger THEN
	        #ts_ErrorText := CONCAT(IN1 := #is_ID, IN2 := ' NORD VFD has internal warning:', IN3 := #ts_ErrorText);
	    END_IF;

	END_REGION

	REGION 5 - Error text german

	    // Clear temorary string
	    #ts_ErrorTextGerman := '';

	    // Possibly error code
	    IF #sx_InternalErrorTrigger OR #sx_InternalWarningTrigger THEN
	        CASE #si_ErrorCode OF
	                // Error code to string code
	            10:
	                #ts_ErrorTextGerman := CONCAT(IN1 := 'Übertemperatur Umrichter, AlarmCode: ', IN2 := #ss_ErrorCode);
	            11:
	                #ts_ErrorTextGerman := CONCAT(IN1 := 'Übertemperatur FU intern, AlarmCode: ', IN2 := #ss_ErrorCode);
	            20:
	                #ts_ErrorTextGerman := CONCAT(IN1 := 'Übertemperatur Motor PTC, AlarmCode: ', IN2 := #ss_ErrorCode);
	            21:
	                #ts_ErrorTextGerman := CONCAT(IN1 := 'Übertemperatur Motor I²t, AlarmCode: ', IN2 := #ss_ErrorCode);
	            22:
	                #ts_ErrorTextGerman := CONCAT(IN1 := 'Übertemperatur Bremswiderstand extern, AlarmCode: ', IN2 := #ss_ErrorCode);
	            30:
	                #ts_ErrorTextGerman := CONCAT(IN1 := 'Überstrom I2t Grenze, AlarmCode: ', IN2 := #ss_ErrorCode);
	            31:
	                #ts_ErrorTextGerman := CONCAT(IN1 := 'Überstrom Chopper , AlarmCode: ', IN2 := #ss_ErrorCode);
	            32:
	                #ts_ErrorTextGerman := CONCAT(IN1 := 'Überstrom IGBT, AlarmCode: ', IN2 := #ss_ErrorCode);
	            33:
	                #ts_ErrorTextGerman := CONCAT(IN1 := 'Überstrom IGBT flink, AlarmCode: ', IN2 := #ss_ErrorCode);
	            40:
	                #ts_ErrorTextGerman := CONCAT(IN1 := 'Überstrom Modul, AlarmCode: ', IN2 := #ss_ErrorCode);
	            41:
	                #ts_ErrorTextGerman := CONCAT(IN1 := 'Überstrom Strommessung, AlarmCode: ', IN2 := #ss_ErrorCode);
	            50:
	                #ts_ErrorTextGerman := CONCAT(IN1 := 'Überspannung UZW, AlarmCode: ', IN2 := #ss_ErrorCode);
	            51:
	                #ts_ErrorTextGerman := CONCAT(IN1 := 'Überspannung Netz, AlarmCode: ', IN2 := #ss_ErrorCode);
	            60:
	                #ts_ErrorTextGerman := CONCAT(IN1 := 'Aufladefehler, AlarmCode: ', IN2 := #ss_ErrorCode);
	            61:
	                #ts_ErrorTextGerman := CONCAT(IN1 := 'Unterspannung Netz, AlarmCode: ', IN2 := #ss_ErrorCode);
	            70:
	                #ts_ErrorTextGerman := CONCAT(IN1 := 'Phasenfehler Netz, AlarmCode: ', IN2 := #ss_ErrorCode);
	            71:
	                #ts_ErrorTextGerman := CONCAT(IN1 := 'Phasenfehler UZW, AlarmCode: ', IN2 := #ss_ErrorCode);
	            80:
	                #ts_ErrorTextGerman := CONCAT(IN1 := 'EEPROM - Maximalwert überschritten, AlarmCode: ', IN2 := #ss_ErrorCode);
	            81:
	                #ts_ErrorTextGerman := CONCAT(IN1 := 'Umrichtertyp falsch, AlarmCode: ', IN2 := #ss_ErrorCode);
	            82:
	                #ts_ErrorTextGerman := CONCAT(IN1 := 'reserviert, AlarmCode: ', IN2 := #ss_ErrorCode);
	            83:
	                #ts_ErrorTextGerman := CONCAT(IN1 := 'EEPROM KSE Fehler, AlarmCode: ', IN2 := #ss_ErrorCode);
	            84:
	                #ts_ErrorTextGerman := CONCAT(IN1 := 'EEPROM interner Fehler, AlarmCode: ', IN2 := #ss_ErrorCode);
	            87:
	                #ts_ErrorTextGerman := CONCAT(IN1 := 'EEPR Kopie ungleich, AlarmCode: ', IN2 := #ss_ErrorCode);
	            100:
	                #ts_ErrorTextGerman := CONCAT(IN1 := 'Bus Time-Out, AlarmCode: ', IN2 := #ss_ErrorCode);
	            101:
	                #ts_ErrorTextGerman := CONCAT(IN1 := 'Systemfehler Option, AlarmCode: ', IN2 := #ss_ErrorCode);
	            102:
	                #ts_ErrorTextGerman := CONCAT(IN1 := 'Bus Time-Out Option, AlarmCode: ', IN2 := #ss_ErrorCode);
	            103:
	                #ts_ErrorTextGerman := CONCAT(IN1 := 'Systemfehler Option, AlarmCode: ', IN2 := #ss_ErrorCode);
	            104:
	                #ts_ErrorTextGerman := CONCAT(IN1 := 'Initfehler Option, AlarmCode: ', IN2 := #ss_ErrorCode);
	            105:
	                #ts_ErrorTextGerman := CONCAT(IN1 := 'Systemfehler Option, AlarmCode: ', IN2 := #ss_ErrorCode);
	            106:
	                #ts_ErrorTextGerman := CONCAT(IN1 := 'Systemfehler Option, AlarmCode: ', IN2 := #ss_ErrorCode);
	            107:
	                #ts_ErrorTextGerman := CONCAT(IN1 := 'Systemfehler Option, AlarmCode: ', IN2 := #ss_ErrorCode);
	            109:
	                #ts_ErrorTextGerman := CONCAT(IN1 := 'Baugruppe fehlt/P120, AlarmCode: ', IN2 := #ss_ErrorCode);
	            110:
	                #ts_ErrorTextGerman := CONCAT(IN1 := 'Kundenschnittstelle, AlarmCode: ', IN2 := #ss_ErrorCode);
	            120:
	                #ts_ErrorTextGerman := CONCAT(IN1 := 'Watchdog extern, AlarmCode: ', IN2 := #ss_ErrorCode);
	            121:
	                #ts_ErrorTextGerman := CONCAT(IN1 := 'Motorische Abschaltgrenze, AlarmCode: ', IN2 := #ss_ErrorCode);
	            122:
	                #ts_ErrorTextGerman := CONCAT(IN1 := 'Generatorische Abschaltgrenze, AlarmCode: ', IN2 := #ss_ErrorCode);
	            123:
	                #ts_ErrorTextGerman := CONCAT(IN1 := 'Drehmomentengrenze, AlarmCode: ', IN2 := #ss_ErrorCode);
	            124:
	                #ts_ErrorTextGerman := CONCAT(IN1 := 'Stromgrenze, AlarmCode: ', IN2 := #ss_ErrorCode);
	            125:
	                #ts_ErrorTextGerman := CONCAT(IN1 := 'Lastmonitor, AlarmCode: ', IN2 := #ss_ErrorCode);
	            128:
	                #ts_ErrorTextGerman := CONCAT(IN1 := 'Analog-In.Minimum, AlarmCode: ', IN2 := #ss_ErrorCode);
	            129:
	                #ts_ErrorTextGerman := CONCAT(IN1 := 'Analog-In.Maximum, AlarmCode: ', IN2 := #ss_ErrorCode);
	            130:
	                #ts_ErrorTextGerman := CONCAT(IN1 := 'Drehgeberfehler, AlarmCode: ', IN2 := #ss_ErrorCode);
	            131:
	                #ts_ErrorTextGerman := CONCAT(IN1 := 'Schleppfehler Drehzahl, AlarmCode: ', IN2 := #ss_ErrorCode);
	            132:
	                #ts_ErrorTextGerman := CONCAT(IN1 := 'Ausschaltüberwachung, AlarmCode: ', IN2 := #ss_ErrorCode);
	            160:
	                #ts_ErrorTextGerman := CONCAT(IN1 := 'Phasenfehler Motor, AlarmCode: ', IN2 := #ss_ErrorCode);
	            161:
	                #ts_ErrorTextGerman := CONCAT(IN1 := 'Magnetisierungsstrom Überwachung, AlarmCode: ', IN2 := #ss_ErrorCode);
	            180:
	                #ts_ErrorTextGerman := CONCAT(IN1 := 'reserviert, AlarmCode: ', IN2 := #ss_ErrorCode);
	            190:
	                #ts_ErrorTextGerman := CONCAT(IN1 := 'Parameteridentifikation, AlarmCode: ', IN2 := #ss_ErrorCode);
	            191:
	                #ts_ErrorTextGerman := CONCAT(IN1 := 'Stern-/ Dreieck-Schaltung Motor falsch, AlarmCode: ', IN2 := #ss_ErrorCode);
	            200:
	                #ts_ErrorTextGerman := CONCAT(IN1 := 'reserviert, AlarmCode: ', IN2 := #ss_ErrorCode);
	            201:
	                #ts_ErrorTextGerman := CONCAT(IN1 := 'Watchdog, AlarmCode: ', IN2 := #ss_ErrorCode);
	            202:
	                #ts_ErrorTextGerman := CONCAT(IN1 := 'Stack Overflow, AlarmCode: ', IN2 := #ss_ErrorCode);
	            203:
	                #ts_ErrorTextGerman := CONCAT(IN1 := 'Stack Underflow, AlarmCode: ', IN2 := #ss_ErrorCode);
	            204:
	                #ts_ErrorTextGerman := CONCAT(IN1 := 'Undefined Opcode, AlarmCode: ', IN2 := #ss_ErrorCode);
	            205:
	                #ts_ErrorTextGerman := CONCAT(IN1 := 'Protected Instruction, AlarmCode: ', IN2 := #ss_ErrorCode);
	            206:
	                #ts_ErrorTextGerman := CONCAT(IN1 := 'Illegal Word Access, AlarmCode: ', IN2 := #ss_ErrorCode);
	            207:
	                #ts_ErrorTextGerman := CONCAT(IN1 := 'Illegal Instruction Access, AlarmCode: ', IN2 := #ss_ErrorCode);
	            208:
	                #ts_ErrorTextGerman := CONCAT(IN1 := 'Programmspeicher Fehler, AlarmCode: ', IN2 := #ss_ErrorCode);
	            209:
	                #ts_ErrorTextGerman := CONCAT(IN1 := 'Dual-Ported RAM, AlarmCode: ', IN2 := #ss_ErrorCode);
	            210:
	                #ts_ErrorTextGerman := CONCAT(IN1 := 'NMI Fehler, AlarmCode: ', IN2 := #ss_ErrorCode);
	            211:
	                #ts_ErrorTextGerman := CONCAT(IN1 := 'PLL Fehler, AlarmCode: ', IN2 := #ss_ErrorCode);
	            212:
	                #ts_ErrorTextGerman := CONCAT(IN1 := 'ADU Fehler, AlarmCode: ', IN2 := #ss_ErrorCode);
	            213:
	                #ts_ErrorTextGerman := CONCAT(IN1 := 'PMI Fehler, AlarmCode: ', IN2 := #ss_ErrorCode);
	            214:
	                #ts_ErrorTextGerman := CONCAT(IN1 := 'Userstack Overflow, AlarmCode: ', IN2 := #ss_ErrorCode);
	            ELSE  // Unknow alarm code
	                #ts_ErrorTextGerman := CONCAT(IN1 := 'Alarm unbekannt, Alarmcode: ', IN2 := #ss_ErrorCode);
	        END_CASE;
	    ELSE
	        #ts_ErrorTextGerman := 'Alarmcode ändern';
	    END_IF;

	    // Write german error code
	    IF #sx_InternalErrorTrigger THEN
	        #ts_ErrorTextGerman := CONCAT(IN1 := #is_ID, IN2 := ' NORD VFD hat interner Fehler: ', IN3 := #ts_ErrorTextGerman);
	    END_IF;

	    IF #sx_InternalWarningTrigger THEN
	        #ts_ErrorTextGerman := CONCAT(IN1 := #is_ID, IN2 := ' NORD VFD hat interner Warnung: ', IN3 := #ts_ErrorTextGerman);
	    END_IF;

	END_REGION

	REGION 6 - Internal VFD Error
	    // Program Alarm internal VFD error
	    #InternalVFDError(SIG := #sx_InternalErrorTrigger,
	                      TIMESTAMP := #Time,
	                      SD_1 := #ts_ErrorText,
	                      SD_2 := #ts_ErrorTextGerman);
	END_REGION

	REGION 7 - Internal VFD Warning
	    // Program Alarm internal VFD Warning
	    #InternalVFDWarning(SIG := #sx_InternalWarningTrigger,
	                        TIMESTAMP := #Time,
	                        SD_1 := #ts_ErrorText,
	                        SD_2 := #ts_ErrorTextGerman);
	END_REGION

	REGION 8 - Profinet slave Error
	    // Program Alarm profinet slave error
	    #PNSlaveError(SIG := #iq_UDT_VFD_Status.PNSlaveError,
	                  TIMESTAMP := #Time,
	                  SD_1 := #is_ID);
	END_REGION

	REGION 9 - Profinet slave not online
	    // Program Alarm profinet slave not online
	    #PNSlaveNotonline(SIG := #iq_UDT_VFD_Status.PNSlaveNotonline,
	                      TIMESTAMP := #Time,
	                      SD_1 := #is_ID);
	END_REGION

	REGION 10 - Profinet slave Error
	    // Program Alarm internal VFD Error
	    #PNSlaveWarnnig(SIG := #iq_UDT_VFD_Status.PNSlaveWarning,
	                    TIMESTAMP := #Time,
	                    SD_1 := #is_ID);
	END_REGION

	REGION 11 - VFD Feedback Error
	    // Program Alarm VFD Feedback Error
	    #VFDRunningFeedbackError(SIG := #iq_UDT_VFD_Status.VFDRunningFeedbackError,
	                             TIMESTAMP := #Time,
	                             SD_1 := #is_ID);
	END_REGION
END_FUNCTION_BLOCK

FUNCTION_BLOCK "FB_TP_ALARM_MFC_Events"
{ S7_Optimized_Access := 'TRUE' }
VERSION : 0.1
// ATTRIBUTES
// AUTO_NUMBER = True
// BLOCK_NUMBER = 182
// END_ATTRIBUTES
   VAR_INPUT
      "Time" { ExternalAccessible := 'False'; ExternalVisible := 'False'; ExternalWritable := 'False'} : LDT;   // Actual Time
      ix_AckHMI { ExternalAccessible := 'False'; ExternalVisible := 'False'; ExternalWritable := 'False'} : Bool;   // Reset
   END_VAR

   VAR_IN_OUT
      iqs_MFCEventsAlarms : "UDT_MFCEvent";   // MFC events alarms structure
   END_VAR

   VAR
      MFCModuleFailure {InstructionName := 'Program_Alarm'; LibVersion := '1.0'; ExternalAccessible := 'False'; ExternalVisible := 'False'; ExternalWritable := 'False'; S7_SetPoint := 'False'} : Program_Alarm;   // MFC Module Failure
      MFCModuleFailureReset {InstructionName := 'Program_Alarm'; LibVersion := '1.0'; ExternalAccessible := 'False'; ExternalVisible := 'False'; ExternalWritable := 'False'; S7_SetPoint := 'False'} : Program_Alarm;   // MFC Module Failure Reset
      MFCNoConnectionToHost {InstructionName := 'Program_Alarm'; LibVersion := '1.0'; ExternalAccessible := 'False'; ExternalVisible := 'False'; ExternalWritable := 'False'; S7_SetPoint := 'False'} : Program_Alarm;   // MFC No Connection To Host
      MFCNoConnectionToHostReset {InstructionName := 'Program_Alarm'; LibVersion := '1.0'; ExternalAccessible := 'False'; ExternalVisible := 'False'; ExternalWritable := 'False'; S7_SetPoint := 'False'} : Program_Alarm;   // MFC No Connection To Host Reset
      MFCNoDestinationFromHost {InstructionName := 'Program_Alarm'; LibVersion := '1.0'; ExternalAccessible := 'False'; ExternalVisible := 'False'; ExternalWritable := 'False'; S7_SetPoint := 'False'} : Program_Alarm;   // MFC No Destination From Host
      MFCNoDestinationFromHostReset {InstructionName := 'Program_Alarm'; LibVersion := '1.0'; ExternalAccessible := 'False'; ExternalVisible := 'False'; ExternalWritable := 'False'; S7_SetPoint := 'False'} : Program_Alarm;   // MFC No Destination From Host Reset
      MFCHostContigency {InstructionName := 'Program_Alarm'; LibVersion := '1.0'; ExternalAccessible := 'False'; ExternalVisible := 'False'; ExternalWritable := 'False'; S7_SetPoint := 'False'} : Program_Alarm;   // MFC Host Contigency
      MFCHostContigencyReset {InstructionName := 'Program_Alarm'; LibVersion := '1.0'; ExternalAccessible := 'False'; ExternalVisible := 'False'; ExternalWritable := 'False'; S7_SetPoint := 'False'} : Program_Alarm;   // MFC Host Contigency Reset
      MFCNoConnectionToHandheldscaner {InstructionName := 'Program_Alarm'; LibVersion := '1.0'; ExternalAccessible := 'False'; ExternalVisible := 'False'; ExternalWritable := 'False'; S7_SetPoint := 'False'} : Program_Alarm;   // MFC No Connection To Handheld scaner
      MFCNoConnectionToHandheldscanerReset {InstructionName := 'Program_Alarm'; LibVersion := '1.0'; ExternalAccessible := 'False'; ExternalVisible := 'False'; ExternalWritable := 'False'; S7_SetPoint := 'False'} : Program_Alarm;   // MFC No Connection To Handheld scaner Reset
      MFCDisableSNCYfinger1 {InstructionName := 'Program_Alarm'; LibVersion := '1.0'; ExternalAccessible := 'False'; ExternalVisible := 'False'; ExternalWritable := 'False'; S7_SetPoint := 'False'} : Program_Alarm;   // MFC Disable SNCY finger 1
      MFCDisableSNCYfinger1Reset {InstructionName := 'Program_Alarm'; LibVersion := '1.0'; ExternalAccessible := 'False'; ExternalVisible := 'False'; ExternalWritable := 'False'; S7_SetPoint := 'False'} : Program_Alarm;   // MFC Disable SNCY finger 1 Reset
      MFCDisableSNCYfinger2 {InstructionName := 'Program_Alarm'; LibVersion := '1.0'; ExternalAccessible := 'False'; ExternalVisible := 'False'; ExternalWritable := 'False'; S7_SetPoint := 'False'} : Program_Alarm;   // MFC Disable SNCY finger 2
      MFCDisableSNCYfinger2Reset {InstructionName := 'Program_Alarm'; LibVersion := '1.0'; ExternalAccessible := 'False'; ExternalVisible := 'False'; ExternalWritable := 'False'; S7_SetPoint := 'False'} : Program_Alarm;   // MFC Disable SNCY finger 2 Reset
      MFCDisableSNCYfinger3 {InstructionName := 'Program_Alarm'; LibVersion := '1.0'; ExternalAccessible := 'False'; ExternalVisible := 'False'; ExternalWritable := 'False'; S7_SetPoint := 'False'} : Program_Alarm;   // MFC Disable SNCY finger 3
      MFCDisableSNCYfinger3Reset {InstructionName := 'Program_Alarm'; LibVersion := '1.0'; ExternalAccessible := 'False'; ExternalVisible := 'False'; ExternalWritable := 'False'; S7_SetPoint := 'False'} : Program_Alarm;   // MFC Disable SNCY finger 3 Reset
      MFCDisableSNCYfinger4 {InstructionName := 'Program_Alarm'; LibVersion := '1.0'; ExternalAccessible := 'False'; ExternalVisible := 'False'; ExternalWritable := 'False'; S7_SetPoint := 'False'} : Program_Alarm;   // MFC Disable SNCY finger 4
      MFCDisableSNCYfinger4Reset {InstructionName := 'Program_Alarm'; LibVersion := '1.0'; ExternalAccessible := 'False'; ExternalVisible := 'False'; ExternalWritable := 'False'; S7_SetPoint := 'False'} : Program_Alarm;   // MFC Disable SNCY finger 4 Reset
      MFCDisableSNCYfinger5 {InstructionName := 'Program_Alarm'; LibVersion := '1.0'; ExternalAccessible := 'False'; ExternalVisible := 'False'; ExternalWritable := 'False'; S7_SetPoint := 'False'} : Program_Alarm;   // MFC Disable SNCY finger 5
      MFCDisableSNCYfinger5Reset {InstructionName := 'Program_Alarm'; LibVersion := '1.0'; ExternalAccessible := 'False'; ExternalVisible := 'False'; ExternalWritable := 'False'; S7_SetPoint := 'False'} : Program_Alarm;   // MFC Disable SNCY finger 5 Reset
   END_VAR


